// TwinCAT 3 PLC project PnpComplexSolution
// ProgramVersion: 3.1.4024.12
// libraries:
//   Tc2_HVAC, * (Beckhoff Automation GmbH)
//   Tc2_MC2, * (Beckhoff Automation GmbH)
//   Tc2_NcKinematicTransformation, * (Beckhoff Automation GmbH)
//   Tc2_Standard, * (Beckhoff Automation GmbH)
//   Tc2_System, * (Beckhoff Automation GmbH)
//   Tc3_Mc3Definitions, * (Beckhoff Automation GmbH)
//   Tc3_McCoordinatedMotion, * (Beckhoff Automation GmbH)
//   Tc3_Module, * (Beckhoff Automation GmbH)
//   VisuSymbols,3.5.10.0,System
// project tree:
//   DUTs/ StructFrame.TcDUT, Xbox.TcDUT
//   / GlobalTextList.TcGTLO, PlcTask.TcTTO, Visualization Manager.TcVMO (not stored)
//   GVLs/ GVL.TcGVL
//   POUs/ FB_AddAllAxes.TcPOU, FB_EnableAxes.TcPOU, FB_NCReset.TcPOU, FB_PowerAll.TcPOU, FrameClass.TcPOU, HMILogic.TcPOU, LoadModel.TcPOU, MAIN.TcPOU, Run.TcPOU, RunXbox.TcPOU
//   VISUs/ Visualization_1.TcVIS
// real-time tasks:
//   TASK PlcTask: cycle T#10ms, priority 20, ADS port 350
//   TASK Job Task: cycle default, priority 32
// motion (NC):
//   TASK NC-Task 1 SAF: cycle T#2ms, priority 4, ADS port 501
//   TASK NC-Task 1 SVB: cycle T#10ms, priority 8, ADS port 511
//   AXIS ACS M1 (id 1)
//     Dynamic: Acceleration=99978.2, Deceleration=99978.2, Jerk=499782000
//     Velo: RefSearch=13.1366666666667, RefSync=13.1366666666667, SlowManual=65.6833333333333, FastManual=394.1, Fast=1313.66666666667
//     OtherSettings: AllowMotionCmdToSlave=true
//     encoder EncType=19
//       EncPara: ScaleFactorNumerator=70, ScaleFactorDenominator=1048576, Offset=-74951.5378, MaxCount=#xffffffff, ReferenceSystem=1
//         SoftEndMinControl: Range=320
//         SoftEndMaxControl: Range=460
//     drive DrvType=16
//       DrvPara: MaxCount=#xffffffff, DriveControlDWord=#x00020100
//         Analog: VeloReferenz=2164.61038933333, VeloScale=32, TorqueSetpointScale=10, ScaleFactorActTorque=0.1
//         TimeComp: TaskDelayCycles=1
//     controller CtrType=1
//       CtrPara: PriorControlFactor=1
//         Observer: BandWidth=20
//   AXIS ACS M2 (id 2)
//     Dynamic: Acceleration=99978.2, Deceleration=99978.2, Jerk=499782000
//     Velo: RefSearch=19.6782762666667, RefSync=19.6782762666667, SlowManual=98.3913813333333, FastManual=590.348288, Fast=1967.82762666667
//     OtherSettings: AllowMotionCmdToSlave=true
//     encoder EncType=19
//       EncPara: ScaleFactorNumerator=104.8576, ScaleFactorDenominator=1048576, Offset=9473.8384, MaxCount=#xffffffff
//     drive DrvType=16
//       DrvPara: MaxCount=#xffffffff, DriveControlDWord=#x00020100
//         Analog: VeloReferenz=2164.61038933333, VeloScale=32, TorqueSetpointScale=10, ScaleFactorActTorque=0.1
//         TimeComp: TaskDelayCycles=1
//     controller CtrType=1
//       CtrPara: PriorControlFactor=1
//         Observer: BandWidth=20
//   AXIS ACS M3 (id 3)
//     Dynamic: Acceleration=99978.2, Deceleration=99978.2, Jerk=499782000
//     Velo: RefSearch=19.6782762666667, RefSync=19.6782762666667, SlowManual=98.3913813333333, FastManual=590.348288, Fast=1967.82762666667
//     OtherSettings: AllowMotionCmdToSlave=true
//     encoder EncType=19
//       EncPara: ScaleFactorNumerator=104.8576, ScaleFactorDenominator=1048576, Offset=-203632.5996, MaxCount=#xffffffff
//     drive DrvType=16
//       DrvPara: MaxCount=#xffffffff, DriveControlDWord=#x00020100
//         Analog: VeloReferenz=2164.61038933333, VeloScale=32, TorqueSetpointScale=10, ScaleFactorActTorque=0.1
//         TimeComp: TaskDelayCycles=1
//     controller CtrType=1
//       CtrPara: PriorControlFactor=1
//         Observer: BandWidth=20
//   AXIS X (id 4)
//     Dynamic: Acceleration=2000, Deceleration=2000, Jerk=2000
//     OtherSettings: AllowMotionCmdToSlave=true
//     encoder EncType=1
//     drive DrvType=5
//       Analog: TorqueSetpointScale=10, ScaleFactorActTorque=0.1
//       TimeComp: TaskDelayCycles=1
//     controller CtrType=1
//       CtrPara: PriorControlFactor=1
//         Observer: BandWidth=20
//   AXIS Y (id 5)
//     Dynamic: Acceleration=2000, Deceleration=2000, Jerk=2000
//     OtherSettings: AllowMotionCmdToSlave=true
//     encoder EncType=1
//     drive DrvType=5
//       Analog: TorqueSetpointScale=10, ScaleFactorActTorque=0.1
//       TimeComp: TaskDelayCycles=1
//     controller CtrType=1
//       CtrPara: PriorControlFactor=1
//         Observer: BandWidth=20
//   AXIS Z (id 6)
//     Dynamic: Acceleration=2000, Deceleration=2000, Jerk=2000
//     OtherSettings: AllowMotionCmdToSlave=true
//     encoder EncType=1
//     drive DrvType=5
//       Analog: TorqueSetpointScale=10, ScaleFactorActTorque=0.1
//       TimeComp: TaskDelayCycles=1
//     controller CtrType=1
//       CtrPara: PriorControlFactor=1
//         Observer: BandWidth=20
// I/O:
//   DEVICE Device 2 (RT-Ethernet Adapter)
//   DEVICE Device 3 (EtherCAT), AmsNetId 192.168.1.168.4.1
//     Box 1 (CU2508) [CU2508 Ethernet Port]
//     Box 2 (EP7211-0034) [EP7211-0034 1Ch. MDP742 Servo motor output stage with OCT (50V, 4.5A RMS)]
//   DEVICE Device 4 (EtherCAT), AmsNetId 192.168.1.168.5.1
//     Box 3 (CU2508) [CU2508 Ethernet Port]
//     Box 4 (EP7211-0034) [EP7211-0034 1Ch. MDP742 Servo motor output stage with OCT (50V, 4.5A RMS)]
//   DEVICE Device 5 (EtherCAT), AmsNetId 192.168.1.168.6.1
//     Box 5 (CU2508) [CU2508 Ethernet Port]
//     Box 6 (EP7211-0034) [EP7211-0034 1Ch. MDP742 Servo motor output stage with OCT (50V, 4.5A RMS)]
//   DEVICE Device 1 (EtherCAT Automation Protocol) (disabled), AmsNetId 192.168.1.168.2.1
//     Box 9 (Publisher)
//     Box 10 (Subscriber)
//   DEVICE Device 6 (EtherCAT), AmsNetId 192.168.1.168.7.1
//     Term 1 (EK1200) [EK1200-5000 EtherCAT Power supply (2A E-Bus)]
//       Term 8 (EL2004) [EL2004 4Ch. Dig. Output 24V, 0.5A]
//       Term 11 (EL1918) [EL1918, 8Ch. Safety Input 24V, TwinSAFE]
//         modules: Module 2 (FSLOGIC)
//       Term 12 (EL2904) [EL2904, 4 Ch. Safety Output 24V, 0.5A, TwinSAFE]
//         modules: Module 1 (FSOES), Module 2 (DO)
//       Term 13 (EL1004) [EL1004 4Ch. Dig. Input 24V, 3ms]
//       Term 14 (EL9512) [EL9512 Power supply terminal 12V]
//       Term 7 (EL9011) [EL9011 End Terminal]
// variable links:
//   Device 6 (EtherCAT) <-> Device 6 (EtherCAT)/Term 1 (EK1200)/Term 12 (EL2904)
//     Term 1 (EK1200)/Term 11 (EL1918)/ConnectionInputs/Message_13 TxPDO <-> Module 1 (FSOES)/RxPDO/FSOE
//     Term 1 (EK1200)/Term 11 (EL1918)/ConnectionOutputs/Message_13 RxPDO <-> Module 1 (FSOES)/TxPDO/FSOE
//   NC-Task 1 SAF/Axes/ACS M1 <-> Device 3 (EtherCAT)/Box 2 (EP7211-0034)
//     Drive/Inputs/In/nDataIn1 <-> DRV Following error actual value/Following error actual value
//     Drive/Inputs/In/nDcOutputTime <-> InfoData/DcOutputShift
//     Drive/Inputs/In/nState1 <-> DRV Statusword/Statusword
//     Drive/Inputs/In/nState2 <-> DRV Statusword/Statusword @bit 8
//     Drive/Inputs/In/nState4 @bit 1 <-> WcState/InputToggle
//     Drive/Inputs/In/nState4 <-> WcState/WcState
//     Drive/Outputs/Out/nCtrl1 <-> DRV Controlword/Controlword
//     Drive/Outputs/Out/nCtrl2 <-> DRV Controlword/Controlword @bit 8
//     Drive/Outputs/Out/nDataOut1 <-> DRV Target position/Target position
//     Enc/Inputs/In/nDataIn1 <-> FB Position/Position
//     Enc/Inputs/In/nDcInputTime <-> InfoData/DcInputShift
//     Enc/Inputs/In/nState4 @bit 1 <-> WcState/InputToggle
//     Enc/Inputs/In/nState4 <-> WcState/WcState
//   NC-Task 1 SAF/Axes/ACS M2 <-> Device 4 (EtherCAT)/Box 4 (EP7211-0034)
//     Drive/Inputs/In/nDataIn1 <-> DRV Following error actual value/Following error actual value
//     Drive/Inputs/In/nDcOutputTime <-> InfoData/DcOutputShift
//     Drive/Inputs/In/nState1 <-> DRV Statusword/Statusword
//     Drive/Inputs/In/nState2 <-> DRV Statusword/Statusword @bit 8
//     Drive/Inputs/In/nState4 @bit 1 <-> WcState/InputToggle
//     Drive/Inputs/In/nState4 <-> WcState/WcState
//     Drive/Outputs/Out/nCtrl1 <-> DRV Controlword/Controlword
//     Drive/Outputs/Out/nCtrl2 <-> DRV Controlword/Controlword @bit 8
//     Drive/Outputs/Out/nDataOut1 <-> DRV Target position/Target position
//     Enc/Inputs/In/nDataIn1 <-> FB Position/Position
//     Enc/Inputs/In/nDcInputTime <-> InfoData/DcInputShift
//     Enc/Inputs/In/nState4 @bit 1 <-> WcState/InputToggle
//     Enc/Inputs/In/nState4 <-> WcState/WcState
//   NC-Task 1 SAF/Axes/ACS M3 <-> Device 5 (EtherCAT)/Box 6 (EP7211-0034)
//     Drive/Inputs/In/nDataIn1 <-> DRV Following error actual value/Following error actual value
//     Drive/Inputs/In/nDcOutputTime <-> InfoData/DcOutputShift
//     Drive/Inputs/In/nState1 <-> DRV Statusword/Statusword
//     Drive/Inputs/In/nState2 <-> DRV Statusword/Statusword @bit 8
//     Drive/Inputs/In/nState4 @bit 1 <-> WcState/InputToggle
//     Drive/Inputs/In/nState4 <-> WcState/WcState
//     Drive/Outputs/Out/nCtrl1 <-> DRV Controlword/Controlword
//     Drive/Outputs/Out/nCtrl2 <-> DRV Controlword/Controlword @bit 8
//     Drive/Outputs/Out/nDataOut1 <-> DRV Target position/Target position
//     Enc/Inputs/In/nDataIn1 <-> FB Position/Position
//     Enc/Inputs/In/nDcInputTime <-> InfoData/DcInputShift
//     Enc/Inputs/In/nState4 @bit 1 <-> WcState/InputToggle
//     Enc/Inputs/In/nState4 <-> WcState/WcState
//   PnpComplexSolution/PnpComplexSolution Instance <-> NC-Task 1 SAF/Axes/ACS M1
//     PlcTask Inputs/GVL.stACSAxis[1].NcToPlc <-> Outputs/ToPlc
//     PlcTask Outputs/GVL.stACSAxis[1].PlcToNc <-> Inputs/FromPlc
//   PnpComplexSolution/PnpComplexSolution Instance <-> NC-Task 1 SAF/Axes/ACS M2
//     PlcTask Inputs/GVL.stACSAxis[2].NcToPlc <-> Outputs/ToPlc
//     PlcTask Outputs/GVL.stACSAxis[2].PlcToNc <-> Inputs/FromPlc
//   PnpComplexSolution/PnpComplexSolution Instance <-> NC-Task 1 SAF/Axes/ACS M3
//     PlcTask Inputs/GVL.stACSAxis[3].NcToPlc <-> Outputs/ToPlc
//     PlcTask Outputs/GVL.stACSAxis[3].PlcToNc <-> Inputs/FromPlc
//   PnpComplexSolution/PnpComplexSolution Instance <-> NC-Task 1 SAF/Axes/X
//     PlcTask Inputs/GVL.stAxis[1].NcToPlc <-> Outputs/ToPlc
//     PlcTask Outputs/GVL.stAxis[1].PlcToNc <-> Inputs/FromPlc
//   PnpComplexSolution/PnpComplexSolution Instance <-> NC-Task 1 SAF/Axes/Y
//     PlcTask Inputs/GVL.stAxis[2].NcToPlc <-> Outputs/ToPlc
//     PlcTask Outputs/GVL.stAxis[2].PlcToNc <-> Inputs/FromPlc
//   PnpComplexSolution/PnpComplexSolution Instance <-> NC-Task 1 SAF/Axes/Z
//     PlcTask Inputs/GVL.stAxis[3].NcToPlc <-> Outputs/ToPlc
//     PlcTask Outputs/GVL.stAxis[3].PlcToNc <-> Inputs/FromPlc
//   PnpComplexSolution/PnpComplexSolution Instance <-> NC-Task 1 SAF/Delta Robot
//     PlcTask Inputs/Run.in_stKinToPlc <-> Outputs/ToPlc
//     PlcTask Outputs/Run.out_stPlcToKin <-> Inputs/FromPlc
//   PnpComplexSolution/PnpComplexSolution Instance <-> NC-Task 1 SAF/Objects/Object1 (MC Group)
//     PlcTask Inputs/GVL.stGroupRef.NcToPlc <-> Group Outputs/ToPLC
//     PlcTask Outputs/GVL.stGroupRef.PlcToNc <-> Group Inputs/FromPLC

CONFIGURATION PnpComplexSolution
    RESOURCE PLC ON TwinCAT3
        TASK PlcTask(INTERVAL := T#10ms, PRIORITY := 20);
        PROGRAM MAIN WITH PlcTask : MAIN;
    END_RESOURCE
END_CONFIGURATION

// ---- DUTs/StructFrame.TcDUT
TYPE StructFrame :
STRUCT
	rXpos : LREAL := 0;
	rYpos : LREAL := 0;
	rZpos : LREAL := 0;
	sAlias : STRING := '';
END_STRUCT
END_TYPE

// ---- DUTs/Xbox.TcDUT
TYPE Xbox :
STRUCT
	bDpadUp : BOOL;
	bDpadDown : BOOL;
	bDpadLeft : BOOL;
	bDpadRight : BOOL;
	
	bXbtn : BOOL;
	bYbtn : BOOL;
	bBbtn : BOOL;
	bAbtn : BOOL;
	
	leftStick : ARRAY [0..2] OF REAL;
	rightStick : ARRAY [0..2] OF REAL;
END_STRUCT
END_TYPE

// ---- GVLs/GVL.TcGVL
VAR_GLOBAL
	stGroupRef			: AXES_GROUP_REF;
	stAxis				: ARRAY[1..cAxesCount] OF AXIS_REF;
	stACSAxis			: ARRAY[1..cAxesCount] OF AXIS_REF;
	PointAPos			: ARRAY[1..5,1..6] OF MC_LREAL;
	PointAPos2			: ARRAY[1..5,1..6] OF MC_LREAL;
	PointBPos			: ARRAY[1..5,1..6] OF MC_LREAL;
	MidPointPos			: ARRAY[1..3] OF MC_LREAL;
	PointAMidPos		: ARRAY[1..3] OF MC_LREAL;
	PointBMidPos		: ARRAY[1..3] OF MC_LREAL;
	PointXTSMidPos		: ARRAY[1..6] OF MC_LREAL;
	PreviousUpPos		: ARRAY[1..3] OF MC_LREAL;
	DeltaVelocity		: INT := 100;
	UpToMidBlend		: INT := 0;
	MidToUpBlend		: INT := 0;
	PointXTSPos			: ARRAY[1..6] OF MC_LREAL;
	
	lrSpeed				: MC_LREAL := 200;
	acceleration		: MC_LREAL := 3000;
END_VAR

VAR_GLOBAL CONSTANT
	cAxesCount			: UINT:=3;
END_VAR

// ---- POUs/MAIN.TcPOU
PROGRAM MAIN
VAR
	init : INT := 0;
	flag : INT := 0;
END_VAR

VAR_INPUT
	bmanual : BOOL;
	bPowerDisable: BOOL;
	bReadDone : BOOL;
END_VAR

HMILogic();
LoadModel();

Run.A_AlwaysActive();

IF bPowerDisable THEN
	Run.A_EnableManualMovement();
	Run.nManual := 0;
	flag := 0;
END_IF

IF bmanual THEN
	Run.A_ReadXYZValue();
	bReadDone := TRUE;
	
END_IF

IF HMILogic.bRun THEN
	IF flag = 0 THEN
		Run.A_EnableManualMovement();
		flag := flag + 1;
	END_IF
	Run(arrangedFrames := HMILogic.ArrangedFrames);
END_IF

END_PROGRAM

// ---- POUs/HMILogic.TcPOU
PROGRAM HMILogic
VAR
	bHmiTeach : BOOL := FALSE;
	bOverride : BOOL := FALSE;

	rCurrentx : LREAL := 0;
	rCurrenty : LREAL := 0;
	rCurrentz : LREAL := 0;
	sCurrentalias : STRING := 'frame';
	
	PRINT : STRING := '';
	
	iCurrentIndex : INT := 0;
	
	iDuplicateIndex : INT := 0;
	
	bThrowHmiException : BOOL := FALSE;
	
	TaughtFrames : ARRAY [0..20] OF StructFrame;
	FrameObject : FrameClass := (AllFrames := TaughtFrames);
	NonEmptyFrames : ARRAY [0..20] OF StructFrame;
	NonEmptyFrameAlias : ARRAY [0..20] OF STRING;
	
	bHmiArrange : BOOL;
	ArrangedAliasInputs : ARRAY [0..20] OF STRING;
	ArrangedIndex : ARRAY[0..20] OF INT;
	ArrangedFrames : ARRAY [0..20] OF StructFrame;
	
	bRun : BOOL := FALSE;
	
	switches : (resting, checkduplicates, handleexception, getframeindex, teachframe, getnonempties);
	bPowerDisable: BOOL;
	bmanual: BOOL;
	bLatch : BOOL;
	iPGT: INT;
	
	XboxController : Xbox;
END_VAR

(*Run.A_EnableManualMovement();
Run.nManual := 0;
IF bPowerDisable THEN
		Run.A_EnableManualMovement();
		bmanual := FALSE;
	END_IF
	
	IF bmanual THEN
		Run.A_ReadXYZValue();
	ELSE
		Run.nManual := 0;
	END_IF*)

(*rCurrentx  := GVL.stAxis[1].NcToPlc.ActPos;
rCurrenty  := GVL.stAxis[2].NcToPlc.ActPos;
rCurrentz  := GVL.stAxis[3].NcToPlc.ActPos;	
Run.A_ReadXYZValue();
	rCurrentx  := GVL.stAxis[1].NcToPlc.ActPos;
	rCurrenty  := GVL.stAxis[2].NcToPlc.ActPos;
	rCurrentz  := GVL.stAxis[3].NcToPlc.ActPos;
*)
	
IF bHmiTeach OR bLatch THEN // if TEACH button is pressed on the HMI
	iPGT := 0;
	
	CASE switches OF
	
		resting: // resting state
			MAIN.bmanual := TRUE;
			IF MAIN.bReadDone THEN
				rCurrentx  := Round2DP(GVL.stAxis[1].NcToPlc.ActPos);
				rCurrenty  := Round2DP(GVL.stAxis[2].NcToPlc.ActPos);
				rCurrentz  := Round2DP(GVL.stAxis[3].NcToPlc.ActPos);
				bLatch := TRUE;
			END_IF
			PRINT := 'RESTING';
			switches := checkduplicates;
			
		checkduplicates: // identify duplicates and throw exception if found
			PRINT := 'CHECKING DUPLICATES';
			iDuplicateIndex := FrameObject.DuplicateExists(sTargetAlias := sCurrentalias); // function returns index of found duplicate, 0 if none are found
			IF iDuplicateIndex = 0 THEN
				switches := getframeindex; // if no duplicates are found, get the first empty frame to teach
			ELSE
				switches := handleexception; // handle the exception
			END_IF
			
		handleexception:
				bThrowHmiException := TRUE; // feedback error to OnButtonUp on the Teach Button to get permission to override
				IF bOverride THEN // if user chooses to override
				PRINT := 'TEACHING FRAMES';
				FrameObject.Teach(iArrayIndex := iDuplicateIndex, rCurrentXpos:= rCurrentx, rCurrentYpos:= rCurrenty,
										rCurrentZpos:= rCurrentz, sAlias:= sCurrentalias); // teach frames
				switches := getnonempties; // filters empty frames
				bOverride := FALSE; // reset variables
				bThrowHmiException := FALSE;
				ELSE
					switches := resting; // filters empty frames
					bHmiTeach := FALSE;
				END_IF
	
		getframeindex:
			PRINT := 'GETTING FRAME INDEX';
			iCurrentIndex := FrameObject.FindFirstEmpty(); // get the first empty frame to teach
			switches := teachframe;
		
		teachframe:
			PRINT := 'TEACHING FRAMES';
			FrameObject.Teach(iArrayIndex := iCurrentIndex, rCurrentXpos:= rCurrentx, rCurrentYpos:= rCurrenty,
	 						rCurrentZpos:= rCurrentz, sAlias:= sCurrentalias); // teach frames
			switches := getnonempties;
		
		getnonempties:
			PRINT := 'GETTING NON EMPTIES';
			NonEmptyFrames := FrameObject.NonEmpty(); // get non-empty frames
			NonEmptyFrameAlias := FrameObject.GetNonEmptyFrameAlias(); // get array of aliases to display in ARRANGE page
			switches := resting;
			bHmiTeach := FALSE;
			MAIN.bmanual := FALSE;
			bLatch := FALSE;
			MAIN.bPowerDisable := TRUE;
	
	END_CASE

ELSIF bRun THEN
	MAIN.bPowerDisable := FALSE;	
	//MAIN.bmanual := TRUE;
	
ELSE
		MAIN.bPowerDisable := TRUE;
END_IF


IF bHmiArrange THEN
	PRINT := 'asasddas';
	ArrangedFrames := FrameObject.MapArrangedAliasToFrameIndex(arrangedAlias := ArrangedAliasInputs, NonEmptyFrames := NonEmptyFrames);
END_IF

METHOD Round2DP : LREAL
VAR_INPUT
	Num : LREAL;
END_VAR
VAR
	meh : INT;
END_VAR
Num := Num * 100;
meh := REAL_TO_INT(Num);
Num := INT_TO_REAL(meh);
Num := Num / 100;
Round2DP := Num;
END_METHOD

END_PROGRAM

// ---- POUs/FrameClass.TcPOU
FUNCTION_BLOCK FrameClass
VAR_INPUT
	AllFrames : ARRAY [0..20] OF StructFrame;
END_VAR
VAR_OUTPUT
END_VAR
VAR
END_VAR

METHOD DuplicateExists : INT
VAR_INPUT
	sTargetAlias : STRING;
END_VAR
VAR
	i : INT;
	n : INT;
END_VAR

FOR i := 0 TO 20 DO
	IF AllFrames[i].sAlias = sTargetAlias THEN
		n := i;
		EXIT;
	ELSE n:=0;
	END_IF
END_FOR

DuplicateExists := n;
END_METHOD

METHOD FindFirstEmpty : INT;
VAR_INPUT
END_VAR
VAR
	EmptyArr : ARRAY[0..20] OF StructFrame;
	i: INT;
	n: INT := 0;
END_VAR
FOR i:=1 TO 20 DO
	IF AllFrames[i].rXpos = 0.0 AND AllFrames[i].rYpos = 0.0 AND AllFrames[i].rZpos = 0.0 AND AllFrames[i].sAlias = '' THEN
		FindFirstEmpty := i;
		EXIT;
	END_IF
END_FOR
END_METHOD

METHOD GetNonEmptyFrameAlias : ARRAY [0..20] OF STRING;
VAR_INPUT
END_VAR
VAR
	i : INT;
	NonEmptyFrames : ARRAY [0..20] OF StructFrame;
	emptyArray : ARRAY [0..20] OF STRING;
END_VAR
NonEmptyFrames := NonEmpty();
FOR i := 0 TO 20 DO
	emptyArray[i] := NonEmptyFrames[i].sAlias;
END_FOR
GetNonEmptyFrameAlias := emptyArray;
END_METHOD

METHOD MapArrangedAliasToFrameIndex : ARRAY[0..20] OF StructFrame;
VAR_INPUT
	arrangedAlias : ARRAY [0..20] OF STRING;
	NonEmptyFrames : ARRAY [0..20] OF StructFrame;
END_VAR

VAR
	mappedArray : ARRAY [0..20] OF StructFrame;
	aliasIndex : INT;
	framesIndex : INT;
	arrangedIndex : INT := 0;
	emptyFrame : StructFrame;
END_VAR
FOR aliasIndex := 0 TO 20 DO
	IF arrangedAlias[aliasIndex] <>  'select' THEN
		FOR framesIndex := 0 TO 20 DO
			IF arrangedAlias[aliasIndex] = NonEmptyFrames[framesIndex].sAlias THEN
				mappedArray[arrangedIndex] := NonEmptyFrames[framesIndex];
				arrangedIndex := arrangedIndex + 1;
				EXIT;
			END_IF
		END_FOR
	ELSE
		mappedArray[arrangedIndex] := emptyFrame;
		arrangedIndex := arrangedIndex + 1;
	END_IF
END_FOR

MapArrangedAliasToFrameIndex := mappedArray;
END_METHOD

METHOD NonEmpty : ARRAY [0..20] OF StructFrame;
VAR_INPUT
END_VAR
VAR
	EmptyArray : ARRAY [0..20] OF StructFrame;
	i : INT;
	n : INT := 0;
END_VAR
FOR i:=1 TO 20 DO
	IF (AllFrames[i].sAlias <> '' ) THEN
		EmptyArray[n] := AllFrames[i];
		n := n+1;
	END_IF
END_FOR
NonEmpty := EmptyArray;
END_METHOD

METHOD Teach : BOOL
VAR_INPUT
	iArrayIndex : INT;
	rCurrentXpos : LREAL;
	rCurrentYpos : LREAL;
	rCurrentZpos : LREAL;
	sAlias : STRING;
END_VAR
VAR
	bSuccess : BOOL := FALSE;
	AugmentedFrame : StructFrame;
END_VAR
AllFrames[iArrayIndex].rXpos := rCurrentXpos;
AllFrames[iArrayIndex].rYpos := rCurrentYpos;
AllFrames[iArrayIndex].rZpos := rCurrentZpos;
AllFrames[iArrayIndex].sAlias := sAlias;
Teach := TRUE;
END_METHOD

END_FUNCTION_BLOCK

// ---- POUs/LoadModel.TcPOU
PROGRAM LoadModel
VAR
	bDone : BOOL;
	iPrediction : INT;
END_VAR

VAR_INPUT
	bPython : BOOL;
END_VAR

IF bPython THEN
	IF bDone THEN
		bPython := FALSE;
		bDone := FALSE;
	END_IF
END_IF

END_PROGRAM

// ---- POUs/Run.TcPOU
PROGRAM Run
VAR	
	buffer					: ARRAY[1..4096] OF BYTE;
	path					: MC_PATH_DATA_REF(ADR(buffer), SIZEOF(buffer));
	
	aTargetPos				: ARRAY[1..cAxesCount] OF MC_LREAL;
	aTransitionParam		: ARRAY[1..2] OF MC_LREAL;
	
	fVelFactor				: LREAL := 1.0;
	
	fbPower					: FB_EnableAxes;
	fbAddAllAxes			: FB_AddAllAxes;
	fbGroupEnable			: MC_GroupEnable;
	fbMoveLinPrep			: MC_MoveLinearAbsolutePreparation;
	fbMovePath				: MC_MovePath;
	fbStop					: MC_GroupStop;
	fbUngroupAxes			: MC_UngroupAllAxes;
	fbGroupReset			: MC_GroupReset;
	fbGroupReadStatus		: MC_GroupReadStatus;
	fbGroupSetOvr			: MC_GroupSetOverride;
	
	nState					: INT := -5;
	nNextState				: INT;
	bMovePrepError			: BOOL;
	bPickCycle				: BOOL;
	bExecutePath			: BOOL := TRUE;
	
	bUserIncrementStep		: BOOL; // user can go to next step
	bUserInfiniteMovement 	: BOOL := TRUE; // user can decide if only one movement is executed or infinite movement.
	bUserStop				: BOOL; // user triggered stop
	bUserForceUngroup		: BOOL; // user triggered ungroup axes
	bUserForceReset			: BOOL; // user triggered reset
	
	
	
	
	bUserEnableAxes:	BOOL:= TRUE;
	bUserConfigGroup:	BOOL	:= FALSE;
	bUserCartesianMode:	BOOL	:= TRUE;
	bUserResetKinGroup:	BOOL	:= FALSE;		
	
	in_stKinToPlc	AT %I*:	NcToPlc_NciChannel_Ref;
	in_stItpToPlc	AT %I*:	NcToPlc_NciChannel_Ref;
	out_stPlcToKin	AT %Q*:	PLCTONC_NCICHANNEL_REF;
	out_stPlcToItp	AT %Q*:	PLCTONC_NCICHANNEL_REF;
	
	//:	FB_EnableAxes;
	bAllAxesReady:	BOOL;
	
	stAxesConfig:	ST_KinAxes;
	fbConfigKinGroup:	FB_KinConfigGroup;
	fbResetKinGroup:	FB_KinResetGroup;
	
	//MODDED CODE VARIABLES
	frameHome : StructFrame := (rXpos := 0, rXpos := 0, rZpos := 147.0, sAlias := 'Home');
	iFrameSequence : INT := 0;
	bRunSequence: BOOL;
	
	
	//////////////
	//Reset
	bResetNC: BOOL;
	bKinFactoryReset: BOOL;
	bResetKinGrp: BOOL;
	nReset: INT;
	nKinReset: INT;
	nGroupReset: INT;
	bKinResetDone: BOOL;
	bGroupResetDone: BOOL;
	fbNCReset	: FB_NCReset;
	bInitMove : BOOL := TRUE;
	iInterpolation : INT := 1;
	bRepeat : BOOL := FALSE;
	
	timerDisable: TON;
	bMagnet: BOOL;
	bXbox : BOOL;
	controller: xbox;
	frameNow: StructFrame;
	frameTarget: StructFrame;
	bAnyBtn : BOOL;
END_VAR

VAR_INPUT
	arrangedFrames : ARRAY [0..20] OF StructFrame;
	nManual: INT;
END_VAR

//==========================================
// PnpSimpleSample V1.3
//==========================================

//==========================================
//	Set variable bUserIncrementStep:= TRUE to go to the next step
//	Variable bUserInfiniteMovement defines if only one movement or infinite
//	movement is executed.
//==========================================



fbGroupReadStatus(
	AxesGroup:= stGroupRef , 
	Enable:= TRUE , 
	Valid=> , 
	Busy=> , 
	GroupMoving=> , 
	GroupHoming=> , 
	GroupErrorStop=> , 
	GroupNotReady=> , 
	GroupStandby=> , 
	GroupStopping=> , 
	GroupDisabled=> , 
	Error=> , 
	ErrorId=> );
IF fbGroupReadStatus.Error THEN
	nState := 9998;
ELSIF NOT fbGroupReadStatus.Valid THEN
	nState := 9999;	
END_IF

fbGroupSetOvr(
	AxesGroup:= stGroupRef, 
	Enable:= TRUE, 
	VelFactor:= fVelFactor , 
	Enabled=> , 
	Busy=> , 
	Error=> , 
	ErrorId=> , 
	ActualVelFactor=> );

IF fbGroupSetOvr.Error THEN
	nState := 9999;
END_IF
	
	


fbPower(
	io_X:= stAxis[1],
	io_Y:= stAxis[2],
	io_Z:= stAxis[3],
	//io_C:= stAxis[4],
	io_M1:= stACSAxis[1],
	io_M2:= stACSAxis[2],
	io_M3:= stACSAxis[3],);
	

stAxesConfig.nAxisIdsAcs[1]	:= stACSAxis[1].NcToPlc.AxisId;
stAxesConfig.nAxisIdsAcs[2]	:= stACSAxis[2].NcToPlc.AxisId;
stAxesConfig.nAxisIdsAcs[3]	:= stACSAxis[3].NcToPlc.AxisId;
stAxesConfig.nAxisIdsMcs[1]	:= stAxis[1].NcToPlc.AxisId;
stAxesConfig.nAxisIdsMcs[2]	:= stAxis[2].NcToPlc.AxisId;
stAxesConfig.nAxisIdsMcs[3]	:= stAxis[3].NcToPlc.AxisId;	
	

CASE nState OF
-5:
	IF bUserIncrementStep THEN
		nNextState := nState +1; 
		nState := 101;
		fbAddAllAxes(Execute:= FALSE);
		fbGroupEnable(AxesGroup:=stGroupRef , Execute:=FALSE);
		fbMovePath(AxesGroup:=stGroupRef ,PathData:=path ,Execute:= FALSE);
		bMovePrepError := FALSE;
	END_IF
-4:	
	fbPower.bEnableAxes := TRUE;
	
	IF fbPower.bAllAxesReady THEN
		IF bUserIncrementStep THEN
			nNextState := nState +1;
			nState := 101;
		END_IF
	ELSIF	fbPower.Error THEN
		nState := nState +1000;	
	END_IF
	
-3:
	fbConfigKinGroup(
		bExecute:=bUserConfigGroup , 
		bCartesianMode:=bUserCartesianMode , 
		stAxesList:=stAxesConfig , 
		stKinRefIn:= in_stKinToPlc, 
		bBusy=> , 
		bDone=> , 
		bError=> , 
		nErrorId=> );
	
	fbResetKinGroup(
		bExecute:=bUserResetKinGroup, 
		nItpChannelId:=0 , 
		stKinRefIn:=in_stKinToPlc, 
		stAxesList:=stAxesConfig, 
		bBusy=> , 
		bDone=> , 
		bError=> , 
		nErrorId=> );
		
	IF fbConfigKinGroup.bDone AND fbResetKinGroup.bDone THEN
		nNextState:= nState + 1;
		nState:= 101;
	ELSIF fbConfigKinGroup.bError OR fbResetKinGroup.bError THEN
		nState:= nState + 1000;
	END_IF
	
-2:
	//Add all axes to group
	fbAddAllAxes(Execute:= TRUE);
	
	IF fbAddAllAxes.Done THEN
		IF bUserIncrementStep THEN
			fbAddAllAxes(Execute:= FALSE);
			nNextState := nState +1;
			nState := 101;
		END_IF
	ELSIF fbAddAllAxes.Error THEN
		nState := nState +1000;
	END_IF
	
-1:	
	//Enable Group
	fbGroupEnable(AxesGroup:=stGroupRef , Execute:=TRUE);
	 
	IF fbGroupEnable.Done THEN
		IF bUserIncrementStep THEN
			fbGroupEnable(AxesGroup:=stGroupRef , Execute:=FALSE);
			nNextState := nState +1;
			nState := 101;
		END_IF
	ELSIF fbGroupEnable.Error THEN
		nState := nState +1000;
	END_IF
0:
	//Fill path table and start execution with fbMovePath
	IF bUserIncrementStep OR bUserInfiniteMovement THEN
		(*IF bPickCycle THEN 
			//Prepare table (MC_MoveLinearAbsolutePreparation)
			A_PreparePathPick();
		ELSE
			//Prepare table (MC_MoveLinearAbsolutePreparation)	
			A_PreparePathPlace();
		END_IF		
		bPickCycle := NOT bPickCycle;*)
		IF bRunSequence THEN
			frameNow.rXpos  := GVL.stAxis[1].NcToPlc.ActPos;
			frameNow.rYpos  := GVL.stAxis[2].NcToPlc.ActPos;
			frameNow.rZpos  := GVL.stAxis[3].NcToPlc.ActPos;
			frameTarget := frameNow;
			END_IF
			
			IF controller.bDpadUp THEN
				//frameTarget := frameNow;
				frameTarget.rYpos := frameNow.rYpos + 1;
				END_IF
			
			IF controller.bDpadDown THEN
				//frameTarget := frameNow;
				frameTarget.rYpos := frameNow.rYpos - 1;
				END_IF
			
			IF controller.bDpadLeft THEN
				//frameTarget := frameNow;
				frameTarget.rXpos := frameNow.rXpos + 1;
				END_IF
			
			IF controller.bDpadRight THEN
				//frameTarget := frameNow;
				frameTarget.rXpos := frameNow.rXpos - 1;
				END_IF
				
			IF controller.bYbtn THEN
				//frameTarget := frameNow;
				frameTarget.rZpos := frameNow.rZpos + 1;
				END_IF
				
			IF controller.bAbtn THEN
				//frameTarget := frameNow;
				frameTarget.rZpos := frameNow.rZpos - 1;
				END_IF
				
			bAnyBtn := (controller.bDpadDown OR controller.bDpadLeft OR controller.bDpadUp OR
						 controller.bDpadRight OR controller.bYbtn OR controller.bAbtn);
			
			IF bAnyBtn THEN
				MoveToPositionGeneral(currentFrame := frameNow, targetFrame := frameTarget, interpolation := 1);
				fbMovePath(AxesGroup:= stGroupRef, PathData:= path, Execute:= TRUE);

				IF bMovePrepError THEN
					nState := nState +1000;
				ELSE
					IF fbMovePath.Done THEN
						fbMovePath(AxesGroup:= stGroupRef, PathData:= path, Execute:= FALSE);
						IF bUserInfiniteMovement THEN
							nState := nState +1;
						ELSIF bUserIncrementStep THEN
							nNextState := nState + 1;
							nState := 101;
						END_IF
					END_IF
				END_IF	
			END_IF			
		END_IF

1:
	//Execute prepared movement
	fbMovePath(
		AxesGroup:= stGroupRef , 
		PathData:= path , 
		Execute:= bExecutePath
	);
	
	IF fbMovePath.Done THEN
		IF bUserIncrementStep THEN
			//ungroup axes
			nNextState := 50;
			nState := 101;
			fbMovePath(AxesGroup:= stGroupRef, PathData:= path, Execute:= FALSE);
		ELSIF bUserInfiniteMovement THEN
			nState := nState -1;
			fbMovePath(AxesGroup:= stGroupRef, PathData:= path, Execute:= FALSE);
		END_IF
	ELSIF fbMovePath.Error THEN
		nState := nState + 1000;	
	END_IF
20:
	fbStop(AxesGroup:=stGroupRef, Execute:= FALSE);
	fbStop(AxesGroup:=stGroupRef, Execute:= TRUE, Jerk:= MC_IGNORE);
	nState := nState + 1;
21:
	fbStop(AxesGroup:=stGroupRef,Execute:= TRUE);
	IF fbStop.Done THEN
		IF bUserIncrementStep THEN
			fbStop(AxesGroup:=stGroupRef, Execute:= FALSE);
			nNextState := 0;
			nState := 101;
		END_IF 		
	ELSIF fbStop.Error THEN
		nState := nState +1000;
	END_IF
50:
	//Disable group and remove all axes 
	fbUngroupAxes(AxesGroup:= stGroupRef, Execute:= FALSE);
	//Check that axes are not moving else we will get a position jump
	IF fbGroupReadStatus.GroupStandby OR fbGroupReadStatus.GroupErrorStop OR fbGroupReadStatus.GroupNotReady THEN
		fbUngroupAxes(AxesGroup:= stGroupRef, Execute:= TRUE);
		nState := nState + 1;
	END_IF	
51:
	fbUngroupAxes(
		AxesGroup:= stGroupRef , 
		Execute:= TRUE, 
		Done=> , 
		Busy=> , 
		Error=> , 
		ErrorId=> );
	
	IF fbUngroupAxes.Done THEN
		IF bUserIncrementStep THEN
			nNextState := -5;
			nState := 101;
		END_IF
	ELSIF fbUngroupAxes.Error THEN
		nState := nState +1000;
	END_IF
80:
	fbGroupReset(AxesGroup:= stGroupRef , Execute:= FALSE);
	fbGroupReset(AxesGroup:= stGroupRef , Execute:= TRUE);
	nState := nState +1;
81:	
	fbGroupReset(
		AxesGroup:= stGroupRef , 
		Execute:= , 
		Done=> , 
		Busy=> , 
		Error=> , 
		ErrorId=> );
	
	IF fbGroupReset.Done THEN
		IF bUserIncrementStep THEN
			IF fbGroupReadStatus.GroupDisabled THEN
				nNextState := -5;
			ELSE
				nNextState := 0;
			END_IF
			nState := 101;
		END_IF				
	END_IF	
101:
	IF (bUserIncrementStep) THEN				
		nState := nNextState;
		bUserIncrementStep := FALSE;
	END_IF
1000..9999:
	;//Error				
END_CASE

IF bUserStop THEN
	nState := 20;
	bUserStop := FALSE;
END_IF
IF bUserForceUngroup THEN
	nState := 50;
	bUserForceUngroup := FALSE;
END_IF
IF bUserForceReset THEN
	nState := 80;
	bUserForceReset := FALSE;
END_IF

ACTION A_AlwaysActive:

fbGroupReadStatus(
	AxesGroup:= stGroupRef , 
	Enable:= TRUE , 
	Valid=> , 
	Busy=> , 
	GroupMoving=> , 
	GroupHoming=> , 
	GroupErrorStop=> , 
	GroupNotReady=> , 
	GroupStandby=> , 
	GroupStopping=> , 
	GroupDisabled=> , 
	Error=> , 
	ErrorId=> );
IF fbGroupReadStatus.Error THEN
	nState := 9998;
ELSIF NOT fbGroupReadStatus.Valid THEN
	nState := 9999;	
END_IF

fbGroupSetOvr(
	AxesGroup:= stGroupRef, 
	Enable:= TRUE, 
	VelFactor:= fVelFactor , 
	Enabled=> , 
	Busy=> , 
	Error=> , 
	ErrorId=> , 
	ActualVelFactor=> );

IF fbGroupSetOvr.Error THEN
	nState := 9999;
END_IF
	
	
fbPower(
	io_X:= stAxis[1],
	io_Y:= stAxis[2],
	io_Z:= stAxis[3],
	io_M1:= stACSAxis[1],
	io_M2:= stACSAxis[2],
	io_M3:= stACSAxis[3]);
	
fbNCReset( 
	bResetDone=> , 
	ResetError=> , 
	io_X:= stAxis[1],     
	io_Y:= stAxis[2],     
	io_Z:= stAxis[3],     
	io_M1:= stACSAxis[1], 
	io_M2:= stACSAxis[2], 
	io_M3:= stACSAxis[3]);	

stAxesConfig.nAxisIdsAcs[1]	:= stACSAxis[1].NcToPlc.AxisId;
stAxesConfig.nAxisIdsAcs[2]	:= stACSAxis[2].NcToPlc.AxisId;
stAxesConfig.nAxisIdsAcs[3]	:= stACSAxis[3].NcToPlc.AxisId;
stAxesConfig.nAxisIdsMcs[1]	:= stAxis[1].NcToPlc.AxisId;
stAxesConfig.nAxisIdsMcs[2]	:= stAxis[2].NcToPlc.AxisId;
stAxesConfig.nAxisIdsMcs[3]	:= stAxis[3].NcToPlc.AxisId;	
	
timerDisable();
END_ACTION

ACTION A_EnableManualMovement:

	fbPower.bEnableAxes := FALSE;
	timerDisable(IN:= TRUE, PT:= T#20MS, Q=> , ET=> );
	IF timerDisable.Q THEN
		fbPower.fOverride := 0;
		fbPower.bEnableAxes := TRUE;
		timerDisable(IN:=FALSE);
		fbNCReset.bReset:=TRUE;
		MAIN.bPowerDisable := FALSE;
	END_IF
END_ACTION

ACTION A_HomePosition:
path.ClearPath();  //Clear nodes that were in path

fbMoveLinPrep.Position						:= ADR(aTargetPos); //pointer to position array
fbMoveLinPrep.PositionCount 				:= cAxesCount; //number of axes in group
fbMoveLinPrep.TransitionParameter			:= ADR (aTransitionParam); //pointer to transition parameter array
fbMoveLinPrep.TransitionParameterCount		:= 2; //number of transition parameters, has to be set always 2
fbMoveLinPrep.BufferMode					:= mcBlendingPrevious;
fbMoveLinPrep.TransitionMode				:= mcTransModeCornerDistanceAdvanced;
//Set dynamics to default values of the axes
fbMoveLinPrep.Acceleration					:= MC_DEFAULT;
fbMoveLinPrep.Deceleration					:= MC_DEFAULT;
fbMoveLinPrep.Jerk							:= MC_DEFAULT;

(* I want to interpolate frames by taking current frame and  next frame,
	and split into N sections, how do i retrieve the current frame? *)

//1st node
aTargetPos[1]				:= 0.0;
aTargetPos[2]				:= 0.0;
aTargetPos[3]				:= 147.0;
////aTargetPos[4]			:= 0;
aTransitionParam[1]			:= 0; //blending distance on previous segment, no influence here
aTransitionParam[2]			:= 0; //blending distance on this segment, no influence here
fbMoveLinPrep(PathData:= path , Velocity:= 200, Acceleration:= 30000, Deceleration:= 30000, Jerk:= 100000, InvokeId:= 10);
bMovePrepError := bMovePrepError OR fbMoveLinPrep.Error;

(*
aTargetPos[1]				:= 100;
aTargetPos[2]				:= 100;
aTargetPos[3]				:= -600;
//aTargetPos[4]			:= 90;
aTransitionParam[1]			:= 30; //blending distance on previous segment (InvokeId=10), defines when to leave line
aTransitionParam[2]			:= 45; //blending distance on this segment, defines latest positionn to be back  on line of InovkeId=20 
fbMoveLinPrep(PathData:= path , Velocity:=200, Acceleration:= 30000, Deceleration:= 30000, Jerk:= 100000, InvokeId:= 20); 
bMovePrepError := bMovePrepError OR fbMoveLinPrep.Error;

aTargetPos[1]				:= 100;
aTargetPos[2]				:= 100;
aTargetPos[3]				:= -750;
//aTargetPos[4]			:= 90;
aTransitionParam[1]			:= 30; 
aTransitionParam[2]			:= 35;
fbMoveLinPrep(PathData:= path , Velocity:= 200, Acceleration:= 30000, Deceleration:= 30000, Jerk:= 100000, InvokeId:= 30);
bMovePrepError := bMovePrepError OR fbMoveLinPrep.Error; *)
END_ACTION

ACTION A_Init:
fbConfigKinGroup(
			bExecute:=FALSE , 
			bCartesianMode:=FALSE , 
			stAxesList:=stAxesConfig , 
			stKinRefIn:= in_stKinToPlc, 
			bBusy=> , 
			bDone=> , 
			bError=> , 
			nErrorId=> );
			
fbResetKinGroup(
			bExecute:=FALSE, 
			nItpChannelId:= , 
			stKinRefIn:=in_stKinToPlc, 
			stAxesList:=stAxesConfig, 
			bBusy=> , 
			bDone=> , 
			bError=> , 
			nErrorId=> );
			
fbNCReset.bReset := FALSE;			
			
bKinResetDone := FALSE;
bGroupResetDone := FALSE;

//bPlace1_Set1 := bPlace2_Set1 := bPlace3_Set1 := bPlace4_Set1:= bPlace5_Set1:= bPlace1_Set2 := bPlace2_Set2 := bPlace3_Set2 := bPlace4_Set2 := FALSE;

//bMagnet_Place1_Set1 := bMagnet_Place2_Set1 := bMagnet_Place3_Set1 := bMagnet_Place1_Set2 := bMagnet_Place2_Set2 := bMagnet_Place3_Set2 := FALSE;
END_ACTION

ACTION A_PreparePathPick:
path.ClearPath();  //Clear nodes that were in path

fbMoveLinPrep.Position						:= ADR(aTargetPos); //pointer to position array
fbMoveLinPrep.PositionCount 				:= cAxesCount; //number of axes in group
fbMoveLinPrep.TransitionParameter			:= ADR (aTransitionParam); //pointer to transition parameter array
fbMoveLinPrep.TransitionParameterCount		:= 2; //number of transition parameters, has to be set always 2
fbMoveLinPrep.BufferMode					:= mcBlendingPrevious;
fbMoveLinPrep.TransitionMode				:= mcTransModeCornerDistanceAdvanced;
//Set dynamics to default values of the axes
fbMoveLinPrep.Acceleration					:= MC_DEFAULT;
fbMoveLinPrep.Deceleration					:= MC_DEFAULT;
fbMoveLinPrep.Jerk							:= MC_DEFAULT;

//1st node
aTargetPos[1]				:= -100;
aTargetPos[2]				:= -100;
aTargetPos[3]				:= -600;
////aTargetPos[4]			:= 0;
aTransitionParam[1]			:= 0; //blending distance on previous segment, no influence here
aTransitionParam[2]			:= 0; //blending distance on this segment, no influence here
fbMoveLinPrep(PathData:= path , Velocity:= 200, Acceleration:= 30000, Deceleration:= 30000, Jerk:= 100000, InvokeId:= 10);
bMovePrepError := bMovePrepError OR fbMoveLinPrep.Error;

aTargetPos[1]				:= 100;
aTargetPos[2]				:= 100;
aTargetPos[3]				:= -600;
////aTargetPos[4]			:= 90;
aTransitionParam[1]			:= 30; //blending distance on previous segment (InvokeId=10), defines when to leave line
aTransitionParam[2]			:= 45; //blending distance on this segment, defines latest positionn to be back  on line of InovkeId=20 
fbMoveLinPrep(PathData:= path , Velocity:=200, Acceleration:= 30000, Deceleration:= 30000, Jerk:= 100000, InvokeId:= 20); 
bMovePrepError := bMovePrepError OR fbMoveLinPrep.Error;

aTargetPos[1]				:= 100;
aTargetPos[2]				:= 100;
aTargetPos[3]				:= -750;
////aTargetPos[4]			:= 90;
aTransitionParam[1]			:= 30; 
aTransitionParam[2]			:= 35;
fbMoveLinPrep(PathData:= path , Velocity:= 200, Acceleration:= 30000, Deceleration:= 30000, Jerk:= 100000, InvokeId:= 30);
bMovePrepError := bMovePrepError OR fbMoveLinPrep.Error;
END_ACTION

ACTION A_PreparePathPlace:
path.ClearPath(); //Clear nodes that were in path

fbMoveLinPrep.Position						:= ADR(aTargetPos); //pointer to position array
fbMoveLinPrep.PositionCount 				:= cAxesCount; //number of axes in group
fbMoveLinPrep.TransitionParameter			:= ADR (aTransitionParam); //pointer to transition parameter array
fbMoveLinPrep.TransitionParameterCount		:= 2; //number of transition parameters, has to be set always 2
fbMoveLinPrep.BufferMode					:= mcBlendingPrevious;
fbMoveLinPrep.TransitionMode				:= mcTransModeCornerDistanceAdvanced;
fbMoveLinPrep.Acceleration					:= MC_DEFAULT;
fbMoveLinPrep.Deceleration					:= MC_DEFAULT;
fbMoveLinPrep.Jerk							:= MC_DEFAULT;

aTargetPos[1]				:= 100;
aTargetPos[2]				:= 100;
aTargetPos[3]				:= -600;
//aTargetPos[4]			:= 90;
aTransitionParam[1]			:= 0; //blending distance on previous segment, no influence here
aTransitionParam[2]			:= 0; //blending distance on this segment, no influence here
fbMoveLinPrep(PathData:= path , Velocity:= 200, Acceleration:= 30000, Deceleration:= 30000, Jerk:= 100000, InvokeId:= 15);
bMovePrepError := bMovePrepError OR fbMoveLinPrep.Error; 

aTargetPos[1]				:= -100;
aTargetPos[2]				:= -100;
aTargetPos[3]				:= -600;
//aTargetPos[4]			:= 0;
aTransitionParam[1]			:= 30; //blending distance on previous segment (InvokeId=10), defines when to leave line
aTransitionParam[2]			:= 45; //blending distance on this segment, defines latest positionn to be back  on line of InovkeId=20
fbMoveLinPrep(PathData:= path , Velocity:= 200, Acceleration:= 30000, Deceleration:= 30000, Jerk:= 100000, InvokeId:= 25);
bMovePrepError := bMovePrepError OR fbMoveLinPrep.Error;

aTargetPos[1]				:= -100;
aTargetPos[2]				:= -100;
aTargetPos[3]				:= -750;
//aTargetPos[4]			:= 0;
aTransitionParam[1]			:= 30; 
aTransitionParam[2]			:= 35;
fbMoveLinPrep(PathData:= path , Velocity:= 200, Acceleration:= 30000, Deceleration:= 30000, Jerk:= 100000, InvokeId:= 35);
bMovePrepError := bMovePrepError OR fbMoveLinPrep.Error;
END_ACTION

ACTION A_ReadXYZValue:
CASE nManual OF
	
	0:
	A_Init();
	nManual := 10;
	bPickCycle := TRUE;
	fbAddAllAxes(Execute:= FALSE);
	fbGroupEnable(AxesGroup:=stGroupRef , Execute:=FALSE);
	fbMovePath(AxesGroup:=stGroupRef ,PathData:=path ,Execute:= FALSE);
	bMovePrepError := FALSE;

10:	
	fbPower.fOverride := 100.0;
	fbPower.bEnableAxes := TRUE;
	
	IF fbPower.bAllAxesReady THEN
		nManual := 20;
	ELSIF	fbPower.Error THEN
		nState := 90;	
	END_IF
	
20:
	bUserConfigGroup:=TRUE;
	bUserCartesianMode:=TRUE;


	fbConfigKinGroup(
		bExecute:=bUserConfigGroup , 
		bCartesianMode:=bUserCartesianMode , 
		stAxesList:=stAxesConfig , 
		stKinRefIn:= in_stKinToPlc, 
		bBusy=> , 
		bDone=> , 
		bError=> , 
		nErrorId=> );
	

	IF fbConfigKinGroup.bDone THEN
		nManual := 100;
	ELSIF fbConfigKinGroup.bError THEN
		nState:= 90;
	END_IF
	(*
30:
	//Add all axes to group
	fbAddAllAxes(Execute:= TRUE);
	
	IF fbAddAllAxes.Done THEN
		fbAddAllAxes(Execute:= FALSE);
		nManual := 40;
	ELSIF fbAddAllAxes.Error THEN
		nState := 90;
	END_IF
	
40:	
	//Enable Group
	fbGroupEnable(AxesGroup:=stGroupRef , Execute:=TRUE);
	 
	IF fbGroupEnable.Done THEN
			fbGroupEnable(AxesGroup:=stGroupRef , Execute:=FALSE);
			nManual := 50;
	ELSIF fbGroupEnable.Error THEN
		nState := 90;
	END_IF
	*)
END_CASE
END_ACTION

METHOD MoveToPositionGeneral
VAR_INPUT
	currentFrame : StructFrame;
	targetFrame : StructFrame;
	interpolation : INT; // interpolates intermittant frames by n number of times
END_VAR

VAR
	unitVector : StructFrame;
	i: INT;
END_VAR
path.ClearPath();  //Clear nodes that were in path

fbMoveLinPrep.Position						:= ADR(aTargetPos); //pointer to position array
fbMoveLinPrep.PositionCount 				:= cAxesCount; //number of axes in group
fbMoveLinPrep.TransitionParameter			:= ADR (aTransitionParam); //pointer to transition parameter array
fbMoveLinPrep.TransitionParameterCount		:= 2; //number of transition parameters, has to be set always 2
fbMoveLinPrep.BufferMode					:= mcBlendingPrevious;
fbMoveLinPrep.TransitionMode				:= mcTransModeCornerDistanceAdvanced;
//Set dynamics to default values of the axes
fbMoveLinPrep.Acceleration					:= MC_DEFAULT;
fbMoveLinPrep.Deceleration					:= MC_DEFAULT;
fbMoveLinPrep.Jerk							:= MC_DEFAULT;

(* I want to interpolate frames by taking current frame and  next frame,
	and split into N sections, how do i retrieve the current frame? *)
	
unitVector.rXpos := (targetFrame.rXpos - currentFrame.rXpos)/interpolation;
unitVector.rYpos := (targetFrame.rYpos - currentFrame.rYpos)/interpolation;
unitVector.rZpos := (targetFrame.rZpos - currentFrame.rZpos)/interpolation;

FOR i:=0 TO interpolation  DO

	//1st node
	aTargetPos[1]				:= currentFrame.rXpos + i * unitVector.rXpos;
	aTargetPos[2]				:= currentFrame.rYpos + i * unitVector.rYpos;
	aTargetPos[3]				:= currentFrame.rZpos + i * unitVector.rZpos;
	//aTargetPos[4]			:= 0;
	aTransitionParam[1]			:= 0; //blending distance on previous segment, no influence here
	aTransitionParam[2]			:= 0; //blending distance on this segment, no influence here
	fbMoveLinPrep(PathData:= path , Velocity:= GVL.lrSpeed, Acceleration:= GVL.acceleration, Deceleration:= GVL.acceleration, Jerk:= 100000, InvokeId:= 30);
	bMovePrepError := bMovePrepError OR fbMoveLinPrep.Error;
	IF bMovePrepError THEN
		EXIT;
	END_IF

END_FOR


(*
aTargetPos[1]				:= 100;
aTargetPos[2]				:= 100;
aTargetPos[3]				:= -600;
//aTargetPos[4]			:= 90;
aTransitionParam[1]			:= 30; //blending distance on previous segment (InvokeId=10), defines when to leave line
aTransitionParam[2]			:= 45; //blending distance on this segment, defines latest positionn to be back  on line of InovkeId=20 
fbMoveLinPrep(PathData:= path , Velocity:=200, Acceleration:= 30000, Deceleration:= 30000, Jerk:= 100000, InvokeId:= 20); 
bMovePrepError := bMovePrepError OR fbMoveLinPrep.Error;

aTargetPos[1]				:= 100;
aTargetPos[2]				:= 100;
aTargetPos[3]				:= -750;
//aTargetPos[4]			:= 90;
aTransitionParam[1]			:= 30; 
aTransitionParam[2]			:= 35;
fbMoveLinPrep(PathData:= path , Velocity:= 200, Acceleration:= 30000, Deceleration:= 30000, Jerk:= 100000, InvokeId:= 30);
bMovePrepError := bMovePrepError OR fbMoveLinPrep.Error; *)
END_METHOD

METHOD MovetoPositionInit
VAR_INPUT
	targetFrame : StructFrame;
END_VAR
path.ClearPath();  //Clear nodes that were in path

fbMoveLinPrep.Position						:= ADR(aTargetPos); //pointer to position array
fbMoveLinPrep.PositionCount 				:= cAxesCount; //number of axes in group
fbMoveLinPrep.TransitionParameter			:= ADR (aTransitionParam); //pointer to transition parameter array
fbMoveLinPrep.TransitionParameterCount		:= 2; //number of transition parameters, has to be set always 2
fbMoveLinPrep.BufferMode					:= mcBlendingPrevious;
fbMoveLinPrep.TransitionMode				:= mcTransModeCornerDistanceAdvanced;
//Set dynamics to default values of the axes
fbMoveLinPrep.Acceleration					:= MC_DEFAULT;
fbMoveLinPrep.Deceleration					:= MC_DEFAULT;
fbMoveLinPrep.Jerk							:= MC_DEFAULT;

(* I want to interpolate frames by taking current frame and  next frame,
	and split into N sections, how do i retrieve the current frame? *)

//1st node
aTargetPos[1]				:= targetFrame.rXpos;
aTargetPos[2]				:= targetFrame.rYpos;
aTargetPos[3]				:= targetFrame.rZpos;
////aTargetPos[4]			:= 0;
aTransitionParam[1]			:= 0; //blending distance on previous segment, no influence here
aTransitionParam[2]			:= 0; //blending distance on this segment, no influence here
fbMoveLinPrep(PathData:= path , Velocity:= GVL.lrSpeed, Acceleration:= GVL.acceleration, Deceleration:= GVL.acceleration, Jerk:= 100000, InvokeId:= 30);
bMovePrepError := bMovePrepError OR fbMoveLinPrep.Error;
END_METHOD

END_PROGRAM

// ---- POUs/FB_EnableAxes.TcPOU
FUNCTION_BLOCK FB_EnableAxes
VAR_INPUT
	bEnableAxes: BOOL:= TRUE;
	fOverride:	LREAL	:= 100.0;
END_VAR
VAR_OUTPUT
	bAllAxesReady:	BOOL:= FALSE;
	Error: BOOL;
END_VAR
VAR_IN_OUT
	io_X:	AXIS_REF;
	io_Y:	AXIS_REF;
	io_Z:	AXIS_REF;
	//io_C:	AXIS_REF;
	io_M1:	AXIS_REF;
	io_M2:	AXIS_REF;
	io_M3:	AXIS_REF;
END_VAR

VAR
	
	fbPowerX:	MC_Power;
	fbPowerY:	MC_Power;
	fbPowerZ:	MC_Power;
	fbPowerC:	MC_Power;
	fbPowerM1:	MC_Power;
	fbPowerM2:	MC_Power;
	fbPowerM3:	MC_Power;
END_VAR

io_X.ReadStatus();
io_Y.ReadStatus();
io_Z.ReadStatus();
//io_C.ReadStatus();
io_M1.ReadStatus();
io_M2.ReadStatus();
io_M3.ReadStatus();


fbPowerX(
	Enable:=bEnableAxes, 
	Enable_Positive:=bEnableAxes, 
	Enable_Negative:=bEnableAxes, 
	Override:=fOverride, 
	BufferMode:= , 
	Axis:=io_X, 
	Status=> , 
	Busy=> , 
	Active=> , 
	Error=> , 
	ErrorID=> );
fbPowerY(
	Enable:=bEnableAxes, 
	Enable_Positive:=bEnableAxes, 
	Enable_Negative:=bEnableAxes, 
	Override:=fOverride, 
	BufferMode:= , 
	Axis:=io_Y, 
	Status=> , 
	Busy=> , 
	Active=> , 
	Error=> , 
	ErrorID=> );	
fbPowerZ(
	Enable:=bEnableAxes, 
	Enable_Positive:=bEnableAxes, 
	Enable_Negative:=bEnableAxes, 
	Override:=fOverride, 
	BufferMode:= , 
	Axis:=io_Z, 
	Status=> , 
	Busy=> , 
	Active=> , 
	Error=> , 
	ErrorID=> );	
(*fbPowerC(
	Enable:=bEnableAxes, 
	Enable_Positive:=bEnableAxes, 
	Enable_Negative:=bEnableAxes, 
	Override:=fOverride, 
	BufferMode:= , 
	Axis:=io_C, 
	Status=> , 
	Busy=> , 
	Active=> , 
	Error=> , 
	ErrorID=> );	*)
fbPowerM1(
	Enable:=bEnableAxes, 
	Enable_Positive:=bEnableAxes, 
	Enable_Negative:=bEnableAxes, 
	Override:=fOverride, 
	BufferMode:= , 
	Axis:=io_M1, 
	Status=> , 
	Busy=> , 
	Active=> , 
	Error=> , 
	ErrorID=> );	
fbPowerM2(
	Enable:=bEnableAxes, 
	Enable_Positive:=bEnableAxes, 
	Enable_Negative:=bEnableAxes, 
	Override:=fOverride, 
	BufferMode:= , 
	Axis:=io_M2, 
	Status=> , 
	Busy=> , 
	Active=> , 
	Error=> , 
	ErrorID=> );	
fbPowerM3(
	Enable:=bEnableAxes, 
	Enable_Positive:=bEnableAxes, 
	Enable_Negative:=bEnableAxes, 
	Override:=fOverride, 
	BufferMode:= , 
	Axis:=io_M3, 
	Status=> , 
	Busy=> , 
	Active=> , 
	Error=> , 
	ErrorID=> );	
bAllAxesReady	:= fbPowerX.Status AND fbPowerY.Status AND fbPowerZ.Status (*AND fbPowerC.Status*) AND 
	fbPowerM1.Status AND fbPowerM2.Status AND fbPowerM3.Status;
	
Error			:= fbPowerX.Error OR fbPowerY.Error OR fbPowerZ.Error OR fbPowerC.Error
	OR fbPowerM1.Error OR fbPowerM2.Error OR fbPowerM3.Error;

END_FUNCTION_BLOCK

// ---- POUs/FB_AddAllAxes.TcPOU
FUNCTION_BLOCK FB_AddAllAxes
VAR_INPUT
	Execute				: BOOL;
END_VAR
VAR_OUTPUT
	Done				: BOOL;
	Busy				: BOOL;
	Error				: BOOL;
END_VAR
VAR
	fbAddAxis			: ARRAY[1..cAxesCount] OF MC_AddAxisToGroup;
	i					: UINT;
END_VAR

Done := TRUE;
Busy := FALSE;
Error := FALSE;

fbAddAxis[1].IdentInGroup := MCS_X; //X-Axis
fbAddAxis[2].IdentInGroup := MCS_Y; //Y-Axis
fbAddAxis[3].IdentInGroup := MCS_Z; //Z-Axis
//fbAddAxis[4].IdentInGroup := MCS_C1;//1st rotation is C-rotation (around Z-Axis)

FOR i:=1 TO cAxesCount DO
	fbAddAxis[i](AxesGroup:=stGroupRef, Axis := stAxis[i], Execute := Execute);

	IF (NOT fbAddAxis[i].Done) THEN
		Done := FALSE;
	END_IF
	IF (fbAddAxis[i].Busy) THEN
		Busy := TRUE;
	END_IF
	IF (fbAddAxis[i].Error) THEN
		Error := TRUE;
	END_IF
END_FOR

END_FUNCTION_BLOCK

// ---- POUs/FB_NCReset.TcPOU
FUNCTION_BLOCK FB_NCReset
VAR_INPUT
	bReset : BOOL;
END_VAR
VAR_OUTPUT
	bResetDone : BOOL;
	ResetError: BOOL;
END_VAR
VAR_IN_OUT
	io_X:	AXIS_REF;
	io_Y:	AXIS_REF;
	io_Z:	AXIS_REF;

	io_M1:	AXIS_REF;
	io_M2:	AXIS_REF;
	io_M3:	AXIS_REF;
	
END_VAR
VAR
	fbResetX : MC_Reset;
	fbResetY : MC_Reset;
	fbResetZ : MC_Reset;
	
	fbResetM1 : MC_Reset;
	fbResetM2 : MC_Reset;
	fbResetM3 : MC_Reset;
END_VAR

fbResetX(
	Axis:= io_X, 
	Execute:= bReset, 
	Done=> , 
	Busy=> , 
	Error=> , 
	ErrorID=> );
	
	fbResetY(
	Axis:= io_Y, 
	Execute:= bReset, 
	Done=> , 
	Busy=> , 
	Error=> , 
	ErrorID=> );
	
	fbResetZ(
	Axis:= io_Z, 
	Execute:= bReset, 
	Done=> , 
	Busy=> , 
	Error=> , 
	ErrorID=> );
	
	fbResetM1(
	Axis:= io_M1, 
	Execute:= bReset, 
	Done=> , 
	Busy=> , 
	Error=> , 
	ErrorID=> );
	
	fbResetM2(
	Axis:= io_M2, 
	Execute:= bReset, 
	Done=> , 
	Busy=> , 
	Error=> , 
	ErrorID=> );
	
	fbResetM3(
	Axis:= io_M3, 
	Execute:= bReset, 
	Done=> , 
	Busy=> , 
	Error=> , 
	ErrorID=> );
	
	
	bResetDone		:= (fbResetX.Done AND fbResetY.Done AND fbResetZ.Done)
	OR (fbResetM1.Done AND fbResetM2.Done AND fbResetM3.Done);
	
	
	ResetError			:= fbResetX.Error OR fbResetY.Error OR fbResetZ.Error
	OR fbResetM1.Error OR fbResetM2.Error OR fbResetM3.Error;

END_FUNCTION_BLOCK

// ---- POUs/FB_PowerAll.TcPOU
FUNCTION_BLOCK FB_PowerAll
VAR_INPUT
	Enable 		: BOOL;
END_VAR
VAR_OUTPUT
	Status		: BOOL;
	Error		: BOOL;
END_VAR
VAR
	fbPower 	: ARRAY [1..cAxesCount] OF MC_Power;
	i			: UINT;
END_VAR

Status := TRUE;
Error := FALSE;

FOR i:=1 TO cAxesCount DO
	fbPower[i](Axis:=stAxis[i],
		Enable			:= Enable,
		Enable_Positive	:= Enable,
		Enable_Negative	:= Enable
	);
	
	Status := Status AND fbPower[i].Status; 
	Error := Error OR fbPower[i].Error;
END_FOR

END_FUNCTION_BLOCK

// ---- POUs/RunXbox.TcPOU
PROGRAM RunXbox
VAR	
	buffer					: ARRAY[1..4096] OF BYTE;
	path					: MC_PATH_DATA_REF(ADR(buffer), SIZEOF(buffer));
	
	aTargetPos				: ARRAY[1..cAxesCount] OF MC_LREAL;
	aTransitionParam		: ARRAY[1..2] OF MC_LREAL;
	
	fVelFactor				: LREAL := 1.0;
	
	fbPower					: FB_EnableAxes;
	fbAddAllAxes			: FB_AddAllAxes;
	fbGroupEnable			: MC_GroupEnable;
	fbMoveLinPrep			: MC_MoveLinearAbsolutePreparation;
	fbMovePath				: MC_MovePath;
	fbStop					: MC_GroupStop;
	fbUngroupAxes			: MC_UngroupAllAxes;
	fbGroupReset			: MC_GroupReset;
	fbGroupReadStatus		: MC_GroupReadStatus;
	fbGroupSetOvr			: MC_GroupSetOverride;
	
	nState					: INT := -5;
	nNextState				: INT;
	bMovePrepError			: BOOL;
	bPickCycle				: BOOL;
	bExecutePath			: BOOL := TRUE;
	
	bUserIncrementStep		: BOOL; // user can go to next step
	bUserInfiniteMovement 	: BOOL := TRUE; // user can decide if only one movement is executed or infinite movement.
	bUserStop				: BOOL; // user triggered stop
	bUserForceUngroup		: BOOL; // user triggered ungroup axes
	bUserForceReset			: BOOL; // user triggered reset
	
	
	
	
	bUserEnableAxes:	BOOL:= TRUE;
	bUserConfigGroup:	BOOL	:= FALSE;
	bUserCartesianMode:	BOOL	:= TRUE;
	bUserResetKinGroup:	BOOL	:= FALSE;		
	
	in_stKinToPlc	AT %I*:	NcToPlc_NciChannel_Ref;
	in_stItpToPlc	AT %I*:	NcToPlc_NciChannel_Ref;
	out_stPlcToKin	AT %Q*:	PLCTONC_NCICHANNEL_REF;
	out_stPlcToItp	AT %Q*:	PLCTONC_NCICHANNEL_REF;
	
	//:	FB_EnableAxes;
	bAllAxesReady:	BOOL;
	
	stAxesConfig:	ST_KinAxes;
	fbConfigKinGroup:	FB_KinConfigGroup;
	fbResetKinGroup:	FB_KinResetGroup;
	
	//MODDED CODE VARIABLES
	frameHome : StructFrame := (rXpos := 0, rXpos := 0, rZpos := 147.0, sAlias := 'Home');
	iFrameSequence : INT := 0;
	bRunSequence: BOOL;
	
	
	//////////////
	//Reset
	bResetNC: BOOL;
	bKinFactoryReset: BOOL;
	bResetKinGrp: BOOL;
	nReset: INT;
	nKinReset: INT;
	nGroupReset: INT;
	bKinResetDone: BOOL;
	bGroupResetDone: BOOL;
	fbNCReset	: FB_NCReset;
	bInitMove : BOOL := TRUE;
	iInterpolation : INT := 5;
	bRepeat : BOOL := FALSE;
	
	timerDisable: TON;
	bMagnet: BOOL;
	
	controller : Xbox;
	rCurrentx: REAL;
	rCurrenty: REAL;
	rCurrentz: REAL;
	frameNow : StructFrame;
	frameTarget : StructFrame;
END_VAR

VAR_INPUT
	arrangedFrames : ARRAY [0..20] OF StructFrame;
	nManual: INT;
END_VAR

//==========================================
// PnpSimpleSample V1.3
//==========================================

//==========================================
//	Set variable bUserIncrementStep:= TRUE to go to the next step
//	Variable bUserInfiniteMovement defines if only one movement or infinite
//	movement is executed.
//==========================================



fbGroupReadStatus(
	AxesGroup:= stGroupRef , 
	Enable:= TRUE , 
	Valid=> , 
	Busy=> , 
	GroupMoving=> , 
	GroupHoming=> , 
	GroupErrorStop=> , 
	GroupNotReady=> , 
	GroupStandby=> , 
	GroupStopping=> , 
	GroupDisabled=> , 
	Error=> , 
	ErrorId=> );
IF fbGroupReadStatus.Error THEN
	nState := 9998;
ELSIF NOT fbGroupReadStatus.Valid THEN
	nState := 9999;	
END_IF

fbGroupSetOvr(
	AxesGroup:= stGroupRef, 
	Enable:= TRUE, 
	VelFactor:= fVelFactor , 
	Enabled=> , 
	Busy=> , 
	Error=> , 
	ErrorId=> , 
	ActualVelFactor=> );

IF fbGroupSetOvr.Error THEN
	nState := 9999;
END_IF
	
	


fbPower(
	io_X:= stAxis[1],
	io_Y:= stAxis[2],
	io_Z:= stAxis[3],
	//io_C:= stAxis[4],
	io_M1:= stACSAxis[1],
	io_M2:= stACSAxis[2],
	io_M3:= stACSAxis[3],);
	

stAxesConfig.nAxisIdsAcs[1]	:= stACSAxis[1].NcToPlc.AxisId;
stAxesConfig.nAxisIdsAcs[2]	:= stACSAxis[2].NcToPlc.AxisId;
stAxesConfig.nAxisIdsAcs[3]	:= stACSAxis[3].NcToPlc.AxisId;
stAxesConfig.nAxisIdsMcs[1]	:= stAxis[1].NcToPlc.AxisId;
stAxesConfig.nAxisIdsMcs[2]	:= stAxis[2].NcToPlc.AxisId;
stAxesConfig.nAxisIdsMcs[3]	:= stAxis[3].NcToPlc.AxisId;	
	

CASE nState OF
-5:
	IF bUserIncrementStep THEN
		nNextState := nState +1; 
		nState := 101;
		fbAddAllAxes(Execute:= FALSE);
		fbGroupEnable(AxesGroup:=stGroupRef , Execute:=FALSE);
		fbMovePath(AxesGroup:=stGroupRef ,PathData:=path ,Execute:= FALSE);
		bMovePrepError := FALSE;
	END_IF
-4:	
	fbPower.bEnableAxes := TRUE;
	
	IF fbPower.bAllAxesReady THEN
		IF bUserIncrementStep THEN
			nNextState := nState +1;
			nState := 101;
		END_IF
	ELSIF	fbPower.Error THEN
		nState := nState +1000;	
	END_IF
	
-3:
	fbConfigKinGroup(
		bExecute:=bUserConfigGroup , 
		bCartesianMode:=bUserCartesianMode , 
		stAxesList:=stAxesConfig , 
		stKinRefIn:= in_stKinToPlc, 
		bBusy=> , 
		bDone=> , 
		bError=> , 
		nErrorId=> );
	
	fbResetKinGroup(
		bExecute:=bUserResetKinGroup, 
		nItpChannelId:=0 , 
		stKinRefIn:=in_stKinToPlc, 
		stAxesList:=stAxesConfig, 
		bBusy=> , 
		bDone=> , 
		bError=> , 
		nErrorId=> );
		
	IF fbConfigKinGroup.bDone AND fbResetKinGroup.bDone THEN
		nNextState:= nState + 1;
		nState:= 101;
	ELSIF fbConfigKinGroup.bError OR fbResetKinGroup.bError THEN
		nState:= nState + 1000;
	END_IF
	
-2:
	//Add all axes to group
	fbAddAllAxes(Execute:= TRUE);
	
	IF fbAddAllAxes.Done THEN
		IF bUserIncrementStep THEN
			fbAddAllAxes(Execute:= FALSE);
			nNextState := nState +1;
			nState := 101;
		END_IF
	ELSIF fbAddAllAxes.Error THEN
		nState := nState +1000;
	END_IF
	
-1:	
	//Enable Group
	fbGroupEnable(AxesGroup:=stGroupRef , Execute:=TRUE);
	 
	IF fbGroupEnable.Done THEN
		IF bUserIncrementStep THEN
			fbGroupEnable(AxesGroup:=stGroupRef , Execute:=FALSE);
			nNextState := nState +1;
			nState := 101;
		END_IF
	ELSIF fbGroupEnable.Error THEN
		nState := nState +1000;
	END_IF
0:
	//Fill path table and start execution with fbMovePath
	IF bUserIncrementStep OR bUserInfiniteMovement THEN
		(*IF bPickCycle THEN 
			//Prepare table (MC_MoveLinearAbsolutePreparation)
			A_PreparePathPick();
		ELSE
			//Prepare table (MC_MoveLinearAbsolutePreparation)	
			A_PreparePathPlace();
		END_IF		
		bPickCycle := NOT bPickCycle;*)
		IF bRunSequence THEN
			
			IF controller.bDpadUp THEN
			frameNow.rXpos  := GVL.stAxis[1].NcToPlc.ActPos;
			frameNow.rYpos  := GVL.stAxis[2].NcToPlc.ActPos;
			frameNow.rZpos  := GVL.stAxis[3].NcToPlc.ActPos;
			
			frameTarget := frameNow;
			frameTarget.rYpos := frameNow.rYpos + 2;
			MoveToPositionGeneral(currentFrame := frameNow, targetFrame := frameTarget, interpolation := 30);
			
			ELSIF controller.bDpadDown THEN
			frameNow.rXpos  := GVL.stAxis[1].NcToPlc.ActPos;
			frameNow.rYpos  := GVL.stAxis[2].NcToPlc.ActPos;
			frameNow.rZpos  := GVL.stAxis[3].NcToPlc.ActPos;
			
			frameTarget := frameNow;
			frameTarget.rYpos := frameNow.rYpos - 2;
			MoveToPositionGeneral(currentFrame := frameNow, targetFrame := frameTarget, interpolation := 30);
			
			ELSIF controller.bDpadLeft THEN
			frameNow.rXpos  := GVL.stAxis[1].NcToPlc.ActPos;
			frameNow.rYpos  := GVL.stAxis[2].NcToPlc.ActPos;
			frameNow.rZpos  := GVL.stAxis[3].NcToPlc.ActPos;
			
			frameTarget := frameNow;
			frameTarget.rXpos := frameNow.rXpos - 2;
			MoveToPositionGeneral(currentFrame := frameNow, targetFrame := frameTarget, interpolation := 30);
			
			ELSIF controller.bDpadRight THEN
			frameNow.rXpos  := GVL.stAxis[1].NcToPlc.ActPos;
			frameNow.rYpos  := GVL.stAxis[2].NcToPlc.ActPos;
			frameNow.rZpos  := GVL.stAxis[3].NcToPlc.ActPos;
			
			frameTarget := frameNow;
			frameTarget.rYpos := frameNow.rXpos + 2;
			MoveToPositionGeneral(currentFrame := frameNow, targetFrame := frameTarget, interpolation := 30);
			

		END_IF
			IF bMovePrepError THEN
				nState := nState +1000;
			ELSE
				fbMovePath(AxesGroup:= stGroupRef, PathData:= path, Execute:= FALSE);
				IF bUserInfiniteMovement THEN
					nState := nState +1;
				ELSIF bUserIncrementStep THEN
					nNextState := nState + 1;
					nState := 101;
				END_IF				
			END_IF	
		END_IF
	END_IF	

1:
	//Execute prepared movement
	fbMovePath(
		AxesGroup:= stGroupRef , 
		PathData:= path , 
		Execute:= bExecutePath
	);
	
	IF fbMovePath.Done THEN
		IF bUserIncrementStep THEN
			//ungroup axes
			nNextState := 50;
			nState := 101;
			fbMovePath(AxesGroup:= stGroupRef, PathData:= path, Execute:= FALSE);
		ELSIF bUserInfiniteMovement THEN
			nState := nState -1;
			fbMovePath(AxesGroup:= stGroupRef, PathData:= path, Execute:= FALSE);
		END_IF
	ELSIF fbMovePath.Error THEN
		nState := nState + 1000;	
	END_IF
20:
	fbStop(AxesGroup:=stGroupRef, Execute:= FALSE);
	fbStop(AxesGroup:=stGroupRef, Execute:= TRUE, Jerk:= MC_IGNORE);
	nState := nState + 1;
21:
	fbStop(AxesGroup:=stGroupRef,Execute:= TRUE);
	IF fbStop.Done THEN
		IF bUserIncrementStep THEN
			fbStop(AxesGroup:=stGroupRef, Execute:= FALSE);
			nNextState := 0;
			nState := 101;
		END_IF 		
	ELSIF fbStop.Error THEN
		nState := nState +1000;
	END_IF
50:
	//Disable group and remove all axes 
	fbUngroupAxes(AxesGroup:= stGroupRef, Execute:= FALSE);
	//Check that axes are not moving else we will get a position jump
	IF fbGroupReadStatus.GroupStandby OR fbGroupReadStatus.GroupErrorStop OR fbGroupReadStatus.GroupNotReady THEN
		fbUngroupAxes(AxesGroup:= stGroupRef, Execute:= TRUE);
		nState := nState + 1;
	END_IF	
51:
	fbUngroupAxes(
		AxesGroup:= stGroupRef , 
		Execute:= TRUE, 
		Done=> , 
		Busy=> , 
		Error=> , 
		ErrorId=> );
	
	IF fbUngroupAxes.Done THEN
		IF bUserIncrementStep THEN
			nNextState := -5;
			nState := 101;
		END_IF
	ELSIF fbUngroupAxes.Error THEN
		nState := nState +1000;
	END_IF
80:
	fbGroupReset(AxesGroup:= stGroupRef , Execute:= FALSE);
	fbGroupReset(AxesGroup:= stGroupRef , Execute:= TRUE);
	nState := nState +1;
81:	
	fbGroupReset(
		AxesGroup:= stGroupRef , 
		Execute:= , 
		Done=> , 
		Busy=> , 
		Error=> , 
		ErrorId=> );
	
	IF fbGroupReset.Done THEN
		IF bUserIncrementStep THEN
			IF fbGroupReadStatus.GroupDisabled THEN
				nNextState := -5;
			ELSE
				nNextState := 0;
			END_IF
			nState := 101;
		END_IF				
	END_IF	
101:
	IF (bUserIncrementStep) THEN				
		nState := nNextState;
		bUserIncrementStep := FALSE;
	END_IF
1000..9999:
	;//Error				
END_CASE

IF bUserStop THEN
	nState := 20;
	bUserStop := FALSE;
END_IF
IF bUserForceUngroup THEN
	nState := 50;
	bUserForceUngroup := FALSE;
END_IF
IF bUserForceReset THEN
	nState := 80;
	bUserForceReset := FALSE;
END_IF

ACTION A_AlwaysActive:

fbGroupReadStatus(
	AxesGroup:= stGroupRef , 
	Enable:= TRUE , 
	Valid=> , 
	Busy=> , 
	GroupMoving=> , 
	GroupHoming=> , 
	GroupErrorStop=> , 
	GroupNotReady=> , 
	GroupStandby=> , 
	GroupStopping=> , 
	GroupDisabled=> , 
	Error=> , 
	ErrorId=> );
IF fbGroupReadStatus.Error THEN
	nState := 9998;
ELSIF NOT fbGroupReadStatus.Valid THEN
	nState := 9999;	
END_IF

fbGroupSetOvr(
	AxesGroup:= stGroupRef, 
	Enable:= TRUE, 
	VelFactor:= fVelFactor , 
	Enabled=> , 
	Busy=> , 
	Error=> , 
	ErrorId=> , 
	ActualVelFactor=> );

IF fbGroupSetOvr.Error THEN
	nState := 9999;
END_IF
	
	
fbPower(
	io_X:= stAxis[1],
	io_Y:= stAxis[2],
	io_Z:= stAxis[3],
	io_M1:= stACSAxis[1],
	io_M2:= stACSAxis[2],
	io_M3:= stACSAxis[3]);
	
fbNCReset( 
	bResetDone=> , 
	ResetError=> , 
	io_X:= stAxis[1],     
	io_Y:= stAxis[2],     
	io_Z:= stAxis[3],     
	io_M1:= stACSAxis[1], 
	io_M2:= stACSAxis[2], 
	io_M3:= stACSAxis[3]);	

stAxesConfig.nAxisIdsAcs[1]	:= stACSAxis[1].NcToPlc.AxisId;
stAxesConfig.nAxisIdsAcs[2]	:= stACSAxis[2].NcToPlc.AxisId;
stAxesConfig.nAxisIdsAcs[3]	:= stACSAxis[3].NcToPlc.AxisId;
stAxesConfig.nAxisIdsMcs[1]	:= stAxis[1].NcToPlc.AxisId;
stAxesConfig.nAxisIdsMcs[2]	:= stAxis[2].NcToPlc.AxisId;
stAxesConfig.nAxisIdsMcs[3]	:= stAxis[3].NcToPlc.AxisId;	
	
timerDisable();
END_ACTION

ACTION A_EnableManualMovement:

	fbPower.bEnableAxes := FALSE;
	timerDisable(IN:= TRUE, PT:= T#20MS, Q=> , ET=> );
	IF timerDisable.Q THEN
		fbPower.fOverride := 0;
		fbPower.bEnableAxes := TRUE;
		timerDisable(IN:=FALSE);
		fbNCReset.bReset:=TRUE;
		MAIN.bPowerDisable := FALSE;
	END_IF
END_ACTION

ACTION A_HomePosition:
path.ClearPath();  //Clear nodes that were in path

fbMoveLinPrep.Position						:= ADR(aTargetPos); //pointer to position array
fbMoveLinPrep.PositionCount 				:= cAxesCount; //number of axes in group
fbMoveLinPrep.TransitionParameter			:= ADR (aTransitionParam); //pointer to transition parameter array
fbMoveLinPrep.TransitionParameterCount		:= 2; //number of transition parameters, has to be set always 2
fbMoveLinPrep.BufferMode					:= mcBlendingPrevious;
fbMoveLinPrep.TransitionMode				:= mcTransModeCornerDistanceAdvanced;
//Set dynamics to default values of the axes
fbMoveLinPrep.Acceleration					:= MC_DEFAULT;
fbMoveLinPrep.Deceleration					:= MC_DEFAULT;
fbMoveLinPrep.Jerk							:= MC_DEFAULT;

(* I want to interpolate frames by taking current frame and  next frame,
	and split into N sections, how do i retrieve the current frame? *)

//1st node
aTargetPos[1]				:= 0.0;
aTargetPos[2]				:= 0.0;
aTargetPos[3]				:= 147.0;
////aTargetPos[4]			:= 0;
aTransitionParam[1]			:= 0; //blending distance on previous segment, no influence here
aTransitionParam[2]			:= 0; //blending distance on this segment, no influence here
fbMoveLinPrep(PathData:= path , Velocity:= 200, Acceleration:= 30000, Deceleration:= 30000, Jerk:= 100000, InvokeId:= 10);
bMovePrepError := bMovePrepError OR fbMoveLinPrep.Error;

(*
aTargetPos[1]				:= 100;
aTargetPos[2]				:= 100;
aTargetPos[3]				:= -600;
//aTargetPos[4]			:= 90;
aTransitionParam[1]			:= 30; //blending distance on previous segment (InvokeId=10), defines when to leave line
aTransitionParam[2]			:= 45; //blending distance on this segment, defines latest positionn to be back  on line of InovkeId=20 
fbMoveLinPrep(PathData:= path , Velocity:=200, Acceleration:= 30000, Deceleration:= 30000, Jerk:= 100000, InvokeId:= 20); 
bMovePrepError := bMovePrepError OR fbMoveLinPrep.Error;

aTargetPos[1]				:= 100;
aTargetPos[2]				:= 100;
aTargetPos[3]				:= -750;
//aTargetPos[4]			:= 90;
aTransitionParam[1]			:= 30; 
aTransitionParam[2]			:= 35;
fbMoveLinPrep(PathData:= path , Velocity:= 200, Acceleration:= 30000, Deceleration:= 30000, Jerk:= 100000, InvokeId:= 30);
bMovePrepError := bMovePrepError OR fbMoveLinPrep.Error; *)
END_ACTION

ACTION A_Init:
fbConfigKinGroup(
			bExecute:=FALSE , 
			bCartesianMode:=FALSE , 
			stAxesList:=stAxesConfig , 
			stKinRefIn:= in_stKinToPlc, 
			bBusy=> , 
			bDone=> , 
			bError=> , 
			nErrorId=> );
			
fbResetKinGroup(
			bExecute:=FALSE, 
			nItpChannelId:= , 
			stKinRefIn:=in_stKinToPlc, 
			stAxesList:=stAxesConfig, 
			bBusy=> , 
			bDone=> , 
			bError=> , 
			nErrorId=> );
			
fbNCReset.bReset := FALSE;			
			
bKinResetDone := FALSE;
bGroupResetDone := FALSE;

//bPlace1_Set1 := bPlace2_Set1 := bPlace3_Set1 := bPlace4_Set1:= bPlace5_Set1:= bPlace1_Set2 := bPlace2_Set2 := bPlace3_Set2 := bPlace4_Set2 := FALSE;

//bMagnet_Place1_Set1 := bMagnet_Place2_Set1 := bMagnet_Place3_Set1 := bMagnet_Place1_Set2 := bMagnet_Place2_Set2 := bMagnet_Place3_Set2 := FALSE;
END_ACTION

ACTION A_PreparePathPick:
path.ClearPath();  //Clear nodes that were in path

fbMoveLinPrep.Position						:= ADR(aTargetPos); //pointer to position array
fbMoveLinPrep.PositionCount 				:= cAxesCount; //number of axes in group
fbMoveLinPrep.TransitionParameter			:= ADR (aTransitionParam); //pointer to transition parameter array
fbMoveLinPrep.TransitionParameterCount		:= 2; //number of transition parameters, has to be set always 2
fbMoveLinPrep.BufferMode					:= mcBlendingPrevious;
fbMoveLinPrep.TransitionMode				:= mcTransModeCornerDistanceAdvanced;
//Set dynamics to default values of the axes
fbMoveLinPrep.Acceleration					:= MC_DEFAULT;
fbMoveLinPrep.Deceleration					:= MC_DEFAULT;
fbMoveLinPrep.Jerk							:= MC_DEFAULT;

//1st node
aTargetPos[1]				:= -100;
aTargetPos[2]				:= -100;
aTargetPos[3]				:= -600;
////aTargetPos[4]			:= 0;
aTransitionParam[1]			:= 0; //blending distance on previous segment, no influence here
aTransitionParam[2]			:= 0; //blending distance on this segment, no influence here
fbMoveLinPrep(PathData:= path , Velocity:= 200, Acceleration:= 30000, Deceleration:= 30000, Jerk:= 100000, InvokeId:= 10);
bMovePrepError := bMovePrepError OR fbMoveLinPrep.Error;

aTargetPos[1]				:= 100;
aTargetPos[2]				:= 100;
aTargetPos[3]				:= -600;
////aTargetPos[4]			:= 90;
aTransitionParam[1]			:= 30; //blending distance on previous segment (InvokeId=10), defines when to leave line
aTransitionParam[2]			:= 45; //blending distance on this segment, defines latest positionn to be back  on line of InovkeId=20 
fbMoveLinPrep(PathData:= path , Velocity:=200, Acceleration:= 30000, Deceleration:= 30000, Jerk:= 100000, InvokeId:= 20); 
bMovePrepError := bMovePrepError OR fbMoveLinPrep.Error;

aTargetPos[1]				:= 100;
aTargetPos[2]				:= 100;
aTargetPos[3]				:= -750;
////aTargetPos[4]			:= 90;
aTransitionParam[1]			:= 30; 
aTransitionParam[2]			:= 35;
fbMoveLinPrep(PathData:= path , Velocity:= 200, Acceleration:= 30000, Deceleration:= 30000, Jerk:= 100000, InvokeId:= 30);
bMovePrepError := bMovePrepError OR fbMoveLinPrep.Error;
END_ACTION

ACTION A_PreparePathPlace:
path.ClearPath(); //Clear nodes that were in path

fbMoveLinPrep.Position						:= ADR(aTargetPos); //pointer to position array
fbMoveLinPrep.PositionCount 				:= cAxesCount; //number of axes in group
fbMoveLinPrep.TransitionParameter			:= ADR (aTransitionParam); //pointer to transition parameter array
fbMoveLinPrep.TransitionParameterCount		:= 2; //number of transition parameters, has to be set always 2
fbMoveLinPrep.BufferMode					:= mcBlendingPrevious;
fbMoveLinPrep.TransitionMode				:= mcTransModeCornerDistanceAdvanced;
fbMoveLinPrep.Acceleration					:= MC_DEFAULT;
fbMoveLinPrep.Deceleration					:= MC_DEFAULT;
fbMoveLinPrep.Jerk							:= MC_DEFAULT;

aTargetPos[1]				:= 100;
aTargetPos[2]				:= 100;
aTargetPos[3]				:= -600;
//aTargetPos[4]			:= 90;
aTransitionParam[1]			:= 0; //blending distance on previous segment, no influence here
aTransitionParam[2]			:= 0; //blending distance on this segment, no influence here
fbMoveLinPrep(PathData:= path , Velocity:= 200, Acceleration:= 30000, Deceleration:= 30000, Jerk:= 100000, InvokeId:= 15);
bMovePrepError := bMovePrepError OR fbMoveLinPrep.Error; 

aTargetPos[1]				:= -100;
aTargetPos[2]				:= -100;
aTargetPos[3]				:= -600;
//aTargetPos[4]			:= 0;
aTransitionParam[1]			:= 30; //blending distance on previous segment (InvokeId=10), defines when to leave line
aTransitionParam[2]			:= 45; //blending distance on this segment, defines latest positionn to be back  on line of InovkeId=20
fbMoveLinPrep(PathData:= path , Velocity:= 200, Acceleration:= 30000, Deceleration:= 30000, Jerk:= 100000, InvokeId:= 25);
bMovePrepError := bMovePrepError OR fbMoveLinPrep.Error;

aTargetPos[1]				:= -100;
aTargetPos[2]				:= -100;
aTargetPos[3]				:= -750;
//aTargetPos[4]			:= 0;
aTransitionParam[1]			:= 30; 
aTransitionParam[2]			:= 35;
fbMoveLinPrep(PathData:= path , Velocity:= 200, Acceleration:= 30000, Deceleration:= 30000, Jerk:= 100000, InvokeId:= 35);
bMovePrepError := bMovePrepError OR fbMoveLinPrep.Error;
END_ACTION

ACTION A_ReadXYZValue:
CASE nManual OF
	
	0:
	A_Init();
	nManual := 10;
	bPickCycle := TRUE;
	fbAddAllAxes(Execute:= FALSE);
	fbGroupEnable(AxesGroup:=stGroupRef , Execute:=FALSE);
	fbMovePath(AxesGroup:=stGroupRef ,PathData:=path ,Execute:= FALSE);
	bMovePrepError := FALSE;

10:	
	fbPower.fOverride := 100.0;
	fbPower.bEnableAxes := TRUE;
	
	IF fbPower.bAllAxesReady THEN
		nManual := 20;
	ELSIF	fbPower.Error THEN
		nState := 90;	
	END_IF
	
20:
	bUserConfigGroup:=TRUE;
	bUserCartesianMode:=TRUE;


	fbConfigKinGroup(
		bExecute:=bUserConfigGroup , 
		bCartesianMode:=bUserCartesianMode , 
		stAxesList:=stAxesConfig , 
		stKinRefIn:= in_stKinToPlc, 
		bBusy=> , 
		bDone=> , 
		bError=> , 
		nErrorId=> );
	

	IF fbConfigKinGroup.bDone THEN
		nManual := 100;
	ELSIF fbConfigKinGroup.bError THEN
		nState:= 90;
	END_IF
	(*
30:
	//Add all axes to group
	fbAddAllAxes(Execute:= TRUE);
	
	IF fbAddAllAxes.Done THEN
		fbAddAllAxes(Execute:= FALSE);
		nManual := 40;
	ELSIF fbAddAllAxes.Error THEN
		nState := 90;
	END_IF
	
40:	
	//Enable Group
	fbGroupEnable(AxesGroup:=stGroupRef , Execute:=TRUE);
	 
	IF fbGroupEnable.Done THEN
			fbGroupEnable(AxesGroup:=stGroupRef , Execute:=FALSE);
			nManual := 50;
	ELSIF fbGroupEnable.Error THEN
		nState := 90;
	END_IF
	*)
END_CASE
END_ACTION

METHOD MoveToPositionGeneral
VAR_INPUT
	currentFrame : StructFrame;
	targetFrame : StructFrame;
	interpolation : INT; // interpolates intermittant frames by n number of times
END_VAR

VAR
	unitVector : StructFrame;
	i: INT;
END_VAR
path.ClearPath();  //Clear nodes that were in path

fbMoveLinPrep.Position						:= ADR(aTargetPos); //pointer to position array
fbMoveLinPrep.PositionCount 				:= cAxesCount; //number of axes in group
fbMoveLinPrep.TransitionParameter			:= ADR (aTransitionParam); //pointer to transition parameter array
fbMoveLinPrep.TransitionParameterCount		:= 2; //number of transition parameters, has to be set always 2
fbMoveLinPrep.BufferMode					:= mcBlendingPrevious;
fbMoveLinPrep.TransitionMode				:= mcTransModeCornerDistanceAdvanced;
//Set dynamics to default values of the axes
fbMoveLinPrep.Acceleration					:= MC_DEFAULT;
fbMoveLinPrep.Deceleration					:= MC_DEFAULT;
fbMoveLinPrep.Jerk							:= MC_DEFAULT;

(* I want to interpolate frames by taking current frame and  next frame,
	and split into N sections, how do i retrieve the current frame? *)
	
unitVector.rXpos := (targetFrame.rXpos - currentFrame.rXpos)/interpolation;
unitVector.rYpos := (targetFrame.rYpos - currentFrame.rYpos)/interpolation;
unitVector.rZpos := (targetFrame.rZpos - currentFrame.rZpos)/interpolation;

FOR i:=0 TO interpolation  DO

	//1st node
	aTargetPos[1]				:= currentFrame.rXpos + i * unitVector.rXpos;
	aTargetPos[2]				:= currentFrame.rYpos + i * unitVector.rYpos;
	aTargetPos[3]				:= currentFrame.rZpos + i * unitVector.rZpos;
	//aTargetPos[4]			:= 0;
	aTransitionParam[1]			:= 0; //blending distance on previous segment, no influence here
	aTransitionParam[2]			:= 0; //blending distance on this segment, no influence here
	fbMoveLinPrep(PathData:= path , Velocity:= GVL.lrSpeed, Acceleration:= GVL.acceleration, Deceleration:= GVL.acceleration, Jerk:= 100000, InvokeId:= 30);
	bMovePrepError := bMovePrepError OR fbMoveLinPrep.Error;
	IF bMovePrepError THEN
		EXIT;
	END_IF

END_FOR


(*
aTargetPos[1]				:= 100;
aTargetPos[2]				:= 100;
aTargetPos[3]				:= -600;
//aTargetPos[4]			:= 90;
aTransitionParam[1]			:= 30; //blending distance on previous segment (InvokeId=10), defines when to leave line
aTransitionParam[2]			:= 45; //blending distance on this segment, defines latest positionn to be back  on line of InovkeId=20 
fbMoveLinPrep(PathData:= path , Velocity:=200, Acceleration:= 30000, Deceleration:= 30000, Jerk:= 100000, InvokeId:= 20); 
bMovePrepError := bMovePrepError OR fbMoveLinPrep.Error;

aTargetPos[1]				:= 100;
aTargetPos[2]				:= 100;
aTargetPos[3]				:= -750;
//aTargetPos[4]			:= 90;
aTransitionParam[1]			:= 30; 
aTransitionParam[2]			:= 35;
fbMoveLinPrep(PathData:= path , Velocity:= 200, Acceleration:= 30000, Deceleration:= 30000, Jerk:= 100000, InvokeId:= 30);
bMovePrepError := bMovePrepError OR fbMoveLinPrep.Error; *)
END_METHOD

METHOD MovetoPositionInit
VAR_INPUT
	targetFrame : StructFrame;
END_VAR
path.ClearPath();  //Clear nodes that were in path

fbMoveLinPrep.Position						:= ADR(aTargetPos); //pointer to position array
fbMoveLinPrep.PositionCount 				:= cAxesCount; //number of axes in group
fbMoveLinPrep.TransitionParameter			:= ADR (aTransitionParam); //pointer to transition parameter array
fbMoveLinPrep.TransitionParameterCount		:= 2; //number of transition parameters, has to be set always 2
fbMoveLinPrep.BufferMode					:= mcBlendingPrevious;
fbMoveLinPrep.TransitionMode				:= mcTransModeCornerDistanceAdvanced;
//Set dynamics to default values of the axes
fbMoveLinPrep.Acceleration					:= MC_DEFAULT;
fbMoveLinPrep.Deceleration					:= MC_DEFAULT;
fbMoveLinPrep.Jerk							:= MC_DEFAULT;

(* I want to interpolate frames by taking current frame and  next frame,
	and split into N sections, how do i retrieve the current frame? *)

//1st node
aTargetPos[1]				:= targetFrame.rXpos;
aTargetPos[2]				:= targetFrame.rYpos;
aTargetPos[3]				:= targetFrame.rZpos;
////aTargetPos[4]			:= 0;
aTransitionParam[1]			:= 0; //blending distance on previous segment, no influence here
aTransitionParam[2]			:= 0; //blending distance on this segment, no influence here
fbMoveLinPrep(PathData:= path , Velocity:= GVL.lrSpeed, Acceleration:= GVL.acceleration, Deceleration:= GVL.acceleration, Jerk:= 100000, InvokeId:= 30);
bMovePrepError := bMovePrepError OR fbMoveLinPrep.Error;
END_METHOD

METHOD Round2DP : LREAL
VAR_INPUT
	Num : LREAL;
END_VAR
VAR
	meh : INT;
END_VAR
Num := Num * 100;
meh := REAL_TO_INT(Num);
Num := INT_TO_REAL(meh);
Num := Num / 100;
Round2DP := Num;
END_METHOD

END_PROGRAM

// ---- GlobalTextList.TcGTLO
TEXTLIST GlobalTextList
  530 = 'Auto '
  903 = 'Disable Power'
  880 = 'Home'
  744 = 'Manual'
  258 = 'Reset'
END_TEXTLIST

// ---- VISUs/Visualization_1.TcVIS
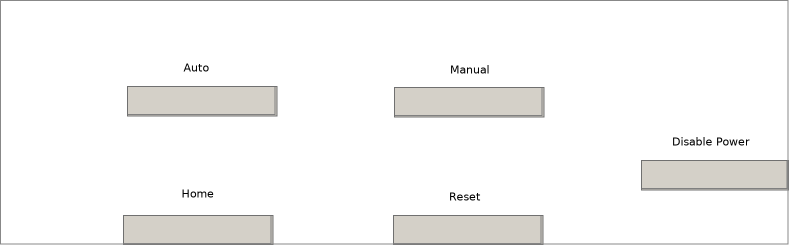
VISUALIZATION Visualization_1  // 789x245
    Button (127,86 150x30)
        tap MAIN.bUserStart
    Button (394,87 150x30)
        tap MAIN.bManual p1329445385=TRUE
    Label (390,182 150x30), "Reset"
    Button (393,215 150x30)
        tap MAIN.bReset
    Button (123,215 150x30)
        tap MAIN.bHome
    Label (123,53 150x30), "Auto"
    Label (123,179 150x30), "Home"
    Label (395,55 150x30), "Manual"
    Label (636,127 150x30), "Disable Power"
    Button (641,160 148x30)
        tap MAIN.bPowerDisable
END_VISUALIZATION
